							Mission^.JPick			:= WorkArea^[Mission^.PPick].JPick + WorkAreaOffset^[Mission^.PPick].J;
							Mission^.KPick			:= Pallet^[Forming^[WorkAreaState^[Mission^.PPlace].F].Pallet].X; (*+ PickPlaceParameters^.OffsetKPick;*)//Layer^[WorkArea^[Mission^.PPick].Layer].X + PickPlaceParameters^.OffsetKPick;//1150;//Layer^[WorkArea^[cwa].Layer].X + 20; 
							Mission^.KPickTorque	:= KPICKTORQUELAYER;
							Mission^.KPickMode 		:= KSUCTIONMODE;
							Mission^.XPlace			:= WorkArea^[Mission^.PPlace].X + WorkAreaOffset^[Mission^.PPlace].X;
							IF WorkAreaState^[cwa].P = 0 THEN       // se devo depositare la falda sul pallet
								Mission^.YPlace			:= WorkArea^[Mission^.PPlace].Y + WorkAreaOffset^[Mission^.PPlace].Y + (Pallet^[Forming^[WorkAreaState^[Mission^.PPlace].F].Pallet].Y / 2); //!!! Modificato !!!!!//WorkArea^[Mission^.PPlace].Y + (Layer^[Forming^[WorkAreaState^[cwa].F].Layer].Y / 2);
								Mission^.ZPlace			:= WorkArea^[Mission^.PPlace].Z + WorkAreaOffset^[Mission^.PPlace].Z + WorkArea^[Mission^.PPlace].H + Layer^[Forming^[WorkAreaState^[Mission^.PPlace].F].Layer].Z + PickPlaceParameters^.OffsetZPlaceLayer;
							ELSE									// se devo depositare la falda su uno strato di pacchi
								Mission^.YPlace			:= WorkArea^[Mission^.PPlace].Y + WorkAreaOffset^[Mission^.PPlace].Y + (Pallet^[Forming^[WorkAreaState^[Mission^.PPlace].F].Pallet].Y / 2);
								Mission^.ZPlace			:= WorkArea^[Mission^.PPlace].H + Layer^[Forming^[WorkAreaState^[Mission^.PPlace].F].PackXP[WorkAreaState^[Mission^.PPlace].P].Layer].Z + PickPlaceParameters^.OffsetZPlaceLayer;
							END_IF
							Mission^.JPlace			:= WorkArea^[Mission^.PPlace].JPlace + WorkAreaOffset^[Mission^.PPlace].J;
							Mission^.KPlace			:= Mission^.KPick;//WorkArea^[Mission^.PPick].KPick;//Layer^[WorkArea^[cwa].Layer].X + 20;
							Mission^.KPlaceMode 	:= KSUCTIONMODE;
							Mission^.XPlaceApproach	:= Mission^.XPlace;
							Mission^.YPlaceApproach	:= Mission^.YPlace;
							Mission^.ZPlaceApproach	:= Mission^.ZPlace;
							Mission^.JPlaceApproach	:= Mission^.JPlace;
							IF WorkAreaState^[Mission^.PPlace].P = 0 THEN			// se devo depositare la falda sul pallet
								Mission^.XDim			:= Layer^[Forming^[WorkAreaState^[Mission^.PPlace].F].Layer].X;
								Mission^.YDim			:= Layer^[Forming^[WorkAreaState^[Mission^.PPlace].F].Layer].Y;
								Mission^.ZDim			:= Layer^[Forming^[WorkAreaState^[Mission^.PPlace].F].Layer].Z;
							ELSE										// se devo depositare la falda su uno strato di pacchi
								Mission^.XDim			:= Layer^[Forming^[WorkAreaState^[Mission^.PPlace].F].PackXP[WorkAreaState^[Mission^.PPlace].P].Layer].X;
								Mission^.YDim			:= Layer^[Forming^[WorkAreaState^[Mission^.PPlace].F].PackXP[WorkAreaState^[Mission^.PPlace].P].Layer].Y;
								Mission^.ZDim			:= Layer^[Forming^[WorkAreaState^[Mission^.PPlace].F].PackXP[WorkAreaState^[Mission^.PPlace].P].Layer].Z;
							END_IF
							
							WorkAreaManager^.State := WAMANAGER_CICLO_PRELIEVO_FALDA_RUN;
							EXIT;
							
						WAMANAGER_CICLO_PRELIEVO_FALDA_RUN:	
							IF Mission^.State = MISSION_STATE_PRELIEVO_FALDA_RUN THEN
								;
							ELSIF Mission^.State = MISSION_STATE_PRELIEVO_FALDA_END THEN
								WorkAreaManager^.State := WAMANAGER_CICLO_PRELIEVO_FALDA_END;
								EXIT;
							ELSIF Mission^.State = MISSION_STATE_ERROR THEN
								;
							END_IF
	
						WAMANAGER_CICLO_PRELIEVO_FALDA_END:	
							//IF Mission^.TPick = TPICK_LAYER THEN
								IF WorkArea^[Mission^.PPick].Typology = TYPOLOGY_LAYER THEN
									IF WorkArea^[Mission^.PPick].H > WorkArea^[Mission^.PPick].Z + Layer^[WorkArea^[Mission^.PPick].Layer].Z THEN
										WorkArea^[Mission^.PPick].H := ModuleAX_Z^.Ax^.Status.ActPosition; (*- WorkArea^[Mission^.PPick].Z;*)//WorkArea^[Mission^.PPick].H - Layer^[WorkArea^[Mission^.PPick].Layer].Z;
										WorkArea^[Mission^.PPick].DoLearn_Z := 2;
										WorkArea^[Mission^.PPick].Learned_Z := ModuleAX_Z^.Ax^.Status.ActPosition;
									ELSE
										WorkArea^[Mission^.PPick].H := 0;
										WorkArea^[Mission^.PPick].DoLearn_Z := 1;
										WorkArea^[Mission^.PPick].Learned_Z := ALTEZZA_CATASTA_FALDE;
										//WorkAreaState^[Mission^.PPick].State := WORKAREA_STATE_OCCUPIED_ENDED;	
									END_IF
								END_IF
							//END_IF
							WorkAreaManager^.State 	:= WAMANAGER_CICLO_DEPOSITO_FALDA_RUN;
							EXIT;
						
						WAMANAGER_CICLO_DEPOSITO_FALDA_RUN:	
							IF Mission^.State = MISSION_STATE_DEPOSITO_FALDA_RUN THEN
								;
							ELSIF Mission^.State = MISSION_STATE_DEPOSITO_FALDA_END THEN
								RestoreCWA^ := TRUE;
								PreviousPWA^ := pwa;
								WorkAreaManager^.State 	:= WAMANAGER_CICLO_DEPOSITO_FALDA_END;	// setto lo stato del WAMANAGER
								EXIT;
							ELSIF Mission^.State = MISSION_STATE_ERROR THEN
								;
							END_IF
							
						WAMANAGER_CICLO_DEPOSITO_FALDA_END:
							//IF WorkAreaState^[Mission^.PPlace].L = 0 THEN						// se la workarea indica l'assenza della falda
								(* Assegno WorkArea^[cwa].L=1 completamento deposito Falda *)
								WorkAreaState^[Mission^.PPlace].L := 1;							// setto la presenza della falda sulla Piazzola dove depositerò il pallet
								WorkAreaState^[Mission^.PPlace].P := WorkAreaState^[Mission^.PPlace].P + 1; // Aggiorno il numero del pacco successivo che si deve depositare
								(* Aggiorno Altezza Pallet su Layer *)
								IF WorkAreaState^[Mission^.PPlace].P > 0 THEN
									WorkArea^[Mission^.PPlace].H := WorkArea^[cwa].H + Layer^[Forming^[WorkAreaState^[Mission^.PPlace].F].Layer].Z;
								ELSE
									WorkArea^[Mission^.PPlace].HPL := WorkArea^[cwa].HPL + Layer^[Forming^[WorkAreaState^[Mission^.PPlace].F].Layer].Z;
								END_IF
								
								(* Aggiorno il numero del pacco successivo che si deve depositare, se il doposito falda è stato effettuato sopra uno strato di pacchi 
								IF WorkAreaState^[Mission^.PPlace].P > 1 THEN						// doposito falda è stato effettuato sopra uno strato di pacchi
										// Aggiorno il numero del pacco successivo che si deve depositare
								ELSE
									WorkAreaState^[Mission^.PPlace].P := 1;							// Aggiorno il numero del pacco successivo che si deve depositare = pacco n°1
								END_IF*)
								
								(* Controllo Fine Pallettizzazione o Deposito Falda Dopo Strato Layer*)
								(* COME FACCIO A SAPERE SE è L'ULTIMO PACCO ? -> Si controlla la Grip=-1 *)
								(* Per sicurezza le controllo su entrambi le direzioni POSITIVA/NEGATIVA *)
								IF Forming^[WorkAreaState^[Mission^.PPlace].F].PackXP[WorkAreaState^[Mission^.PPlace].P].Grip = -1 OR
									Forming^[WorkAreaState^[Mission^.PPlace].F].PackXN[WorkAreaState^[Mission^.PPlace].P].Grip = -1 THEN
									WorkAreaState^[Mission^.PPlace].State := WORKAREA_STATE_OCCUPIED_WORKED;
								END_IF	
								
								RestoreCWA^ := TRUE;
								PreviousPWA^ := pwa;
								WorkAreaManager^.State 	:= WAMANAGER_NOP;
								EXIT;	
							//ELSE														// non dovrebbe mai accadere
							//	WorkAreaState^[cwa].L := 1;	
							//	WorkAreaState^[cwa].State := WORKAREA_STATE_OCCUPIED_WORKED;
							//	WorkAreaManager^.State 	:= WAMANAGER_NOP;
							//	EXIT;
							//END_IF
							
						(* Creo Missione Pacco *)
						WAMANAGER_CICLO_PACCO_INIT:
							IF cwa = UltimaWAAssegnazionePacco AND cwa<>0 THEN
								(* Reset della memoria utilizzata per forzare il ciclo di riposo in ciclo di prelievo pacco *)
								//ForzaPrelievoPaccoDuranteCicloDiRiposo := FALSE;			
								(* Definisco dse la WORKAREA è negativa o positiva *)
								IF WorkAreaState^[cwa].PN < 0 THEN							// se la Workarea non è stata inizializzata (-1) vado a definire se è a DX o SX del ribaltino
									IF WorkPickPoint^[ppick].Xv < WorkArea^[cwa].X THEN		// Se la quota X è MINORE della quota del ribaltino definisco che la workarea è NEGATIVA 
										WorkAreaState^[cwa].PN := 0;
									ELSE													// Se la quota X è MAGGIORE della quota del ribaltino definisco che la workarea è POSITIVA 
										WorkAreaState^[cwa].PN := 1;
									END_IF
								END_IF
								
								Mission^.PPick := ppick;								   	// Assegno il numero della Punto di prelievo
								Mission^.TPick := TPICK_PACK;							   	// Assegno il tipo di Prelievo
								Mission^.PPlace := cwa;									   	// Assegno il numero della piazzola di deposito
								Mission^.XDim := WorkPickPointState^[Mission^.PPick].XDim; 	// Assegno la dimensione X del pacco presente nel punto di prelievo designato
								Mission^.YDim := WorkPickPointState^[Mission^.PPick].YDim; 	// Assegno la dimensione X del pacco presente nel punto di prelievo designato
								Mission^.ZDim := WorkPickPointState^[Mission^.PPick].ZDim; 	// Assegno la dimensione X del pacco presente nel punto di prelievo designato
								
								(* Definisco il tipo di presa dei pacchi "sinistri" e "destri" *)
								IF WorkAreaState^[cwa].PN = 0 THEN							
									jp := Forming^[WorkAreaState^[cwa].F].PackXP[WorkAreaState^[cwa].P].JP;		// Tipo di presa della pinza
									vo := Forming^[WorkAreaState^[cwa].F].PackXP[WorkAreaState^[cwa].P].Grip;	// Tipo di disposizione del pacco sul ribaltino
								ELSE
									jp := Forming^[WorkAreaState^[cwa].F].PackXN[WorkAreaState^[cwa].P].JP;		// Tipo di presa della pinza
									vo := Forming^[WorkAreaState^[cwa].F].PackXN[WorkAreaState^[cwa].P].Grip;	// Tipo di disposizione del pacco sul ribaltino
								END_IF
								(* Controllo se lo spessore del pacco è minore della lunghezza della pinza *)
								IF Mission^.ZDim < TCPParameter^.Z AND 						// Altezza pacco sul ribaltino < di un parametro
									vo = 1 THEN												// Presa pacco in orrizzontale
									ZOffsetPick 	:= TCPParameter^.Z - Mission^.ZDim;		// Offset da utilizzare successivamente nel calcolo della quota di prelievo
									ZOffsetPlace 	:= TCPParameter^.Z - Mission^.ZDim;		// Offset da utilizzare successivamente nel calcolo della quota di prelievo
								ELSE	
									ZOffsetPick 	:= 0;									// Offset da utilizzare successivamente nel calcolo della quota di prelievo
									ZOffsetPlace 	:= 0;									// Offset da utilizzare successivamente nel calcolo della quota di prelievo
								END_IF
								
								IF vo = 0 THEN 															// Se ho prelievo verticale
									CASE TIPO_RIBALTINO OF
										(* TIPO 1 = RIBALTINO_DOPO_SQUADRO *)
										1: 
											HalfPackDim := Mission^.YDim/2;										// Metà pacco = (dimensione Y)/2
											(* Verticale *)
											IF jp = 1 THEN														// Prelievo lungo X (Longitudinale)
												(* Longitudinale *)
												kpick := Mission^.XDim;										 	// Quota di prelievo Asse K
												torque := Forming^[WorkAreaState^[cwa].F].KLT;					// Valore di coppia Asse K
											ELSE																// Prelievo lungo Y (Trasversale)
												(* Trasversale *)
												kpick := Mission^.ZDim;	//Forming^[WorkAreaState^[cwa].F].PZ;	// Quota di prelievo Asse K
												torque := Forming^[WorkAreaState^[cwa].F].KTT;					// Valore di coppia Asse K
											END_IF
											XPick := WorkPickPoint^[Mission^.PPick].Xv + 		// Quota X Ribaltino
													 WorkPickPointOffset^[Mission^.PPick].Xv;	//Offset Posizione ribaltino in direzione X	
											YPick := WorkPickPoint^[Mission^.PPick].Yv + 		// Quota Y ribaltino
													 WorkPickPointOffset^[Mission^.PPick].Yv + //Offset Posizione ribaltino in direzione Y
													 (Mission^.ZDim / 2);					// (Dimensione pacco Z)/2
											ZPick := WorkPickPoint^[Mission^.PPick].Zv + 	// Quota Z ribaltino
													 WorkPickPointOffset^[Mission^.PPick].Zv + //Offset Posizione ribaltino in direzione Z	
													 Mission^.YDim + 						// Dimensione Y del pacco	
													 Forming^[WorkAreaState^[cwa].F].PIZ + 	// Offset di prelievo dato dalla formatura			
													 WorkPickPointState^[ppick].ZTilter;	// Quota asse ribaltino
											(* In base al tipo di pallettizzatore setto la quota per la presa in modo che i pacchi vengano depositati in modo corretto *)		 		 
											CASE VERSO_PALLETTIZZATORE OF
												PALLETTIZZATORE_DX:
																	JPick := WorkPickPoint^[Mission^.PPick].Jv + 		// Quota rotazione data dalla disposizione del ribaltino
																			 WorkPickPointOffset^[Mission^.PPick].Jv + 	//Offset Posizione ribaltino in direzione Z	
																 			(90 * jp) - 90 +							// Quota rotazione stabilita dal tipo di presa	
																			180;
											
												PALLETTIZZATORE_SX:
																	JPick := WorkPickPoint^[Mission^.PPick].Jv + 	// Quota rotazione data dalla disposizione del ribaltino
																			 WorkPickPointOffset^[Mission^.PPick].Jv + //Offset Posizione ribaltino in direzione Z	
																 			(90 * jp) - 90;								// Quota rotazione stabilita dal tipo di presa								
											END_CASE		 
											(* Differenza tra valori reali e nominali  *)
											DifferenceRealNominalDimensionZ := Mission^.YDim - Forming^[WorkAreaState^[cwa].F].PY;
											(* Valorizzo la variabile che serve per calolare la quota di fuori ingombro verticale della pinza *)
											Dimensione_Z_ElementoInPresaX_Ingombro := Mission^.YDim + Forming^[WorkAreaState^[cwa].F].PIZ;
										(* TIPO 2 = RIBALTINO_DIRETTO *)
										2:
											HalfPackDim := Mission^.ZDim/2;										// Metà pacco = (dimensione Z)/2
											(* Verticale *)
											IF jp = 0 THEN														// Prelievo (Longitudinale)
												(* Longitudinale *)
												kpick := Mission^.ZDim;                                     	// Quota di prelievo Asse K
												torque := Forming^[WorkAreaState^[cwa].F].KLT;					// Valore di coppia Asse K
											ELSE																// Prelievo lungo Y (Trasversale)
												(* Trasversale *)
												kpick := Mission^.YDim;	//Forming^[WorkAreaState^[cwa].F].PZ;	// Quota di prelievo Asse K
												torque := Forming^[WorkAreaState^[cwa].F].KTT;					// Valore di coppia Asse K
											END_IF
											XPick := WorkPickPoint^[Mission^.PPick].Xv + 		// Quota X Ribaltino
													 WorkPickPointOffset^[Mission^.PPick].Xv +	//Offset Posizione ribaltino in direzione X	
													 Mission^.ZDim/2;								// Metà pacco = (dimensione Z) /2
											YPick := WorkPickPoint^[Mission^.PPick].Yv + 		// Quota Y ribaltino
													 WorkPickPointOffset^[Mission^.PPick].Yv;  //Offset Posizione ribaltino in direzione Y
													//(Mission^.ZDim / 2);					// (Dimensione pacco Z)/2
											ZPick := WorkPickPoint^[Mission^.PPick].Zv + 	// Quota Z ribaltino
													 WorkPickPointOffset^[Mission^.PPick].Zv + //Offset Posizione ribaltino in direzione Z	
													 Mission^.XDim + 						// Dimensione Y del pacco	
													 Forming^[WorkAreaState^[cwa].F].PIZ + 	// Offset di prelievo dato dalla formatura			
													 WorkPickPointState^[ppick].ZTilter;	// Quota asse ribaltino
											(* In base al tipo di pallettizzatore setto la quota per la presa in modo che i pacchi vengano depositati in modo corretto *)		 
											CASE VERSO_PALLETTIZZATORE OF
												PALLETTIZZATORE_DX:
																	JPick := WorkPickPoint^[Mission^.PPick].Jv + 	// Quota rotazione data dalla disposizione del ribaltino
																			 WorkPickPointOffset^[Mission^.PPick].Jv + //Offset Posizione ribaltino in direzione Z	
														 					(90 * (1-jp))+								// Quota rotazione stabilita dal tipo di presa	
																			180;										// +180° per fare in modo che il deposito sul pallet sia uguale per le formature con verso del pal DX e SX
												
												PALLETTIZZATORE_SX:	
																	JPick := WorkPickPoint^[Mission^.PPick].Jv + 	// Quota rotazione data dalla disposizione del ribaltino
																			 WorkPickPointOffset^[Mission^.PPick].Jv + //Offset Posizione ribaltino in direzione Z	
														 					(90 * (1-jp));								// Quota rotazione stabilita dal tipo di presa							
											END_CASE
											(* Differenza tra valori reali e nominali  *)
											DifferenceRealNominalDimensionZ := Mission^.XDim - Forming^[WorkAreaState^[cwa].F].PY;
											(* Valorizzo la variabile che serve per calolare la quota di fuori ingombro verticale della pinza *)
											Dimensione_Z_ElementoInPresaX_Ingombro := Mission^.XDim + Forming^[WorkAreaState^[cwa].F].PIZ;
									END_CASE
									
								ELSE																	// Se ho prelievo orrizzontale
									CASE TIPO_RIBALTINO OF
										(* TIPO 1 = RIBALTINO_DOPO_SQUADRO *)
										1:
											HalfPackDim := Mission^.ZDim/2; 									// Metà pacco = (dimensione Z) /2
											(* Orizzontale *)
											IF jp = 1 THEN														// Prelievo TRASVERSALE
												(* Trasversale *)
												kpick := Mission^.XDim; 										 // Quota di prelievo Asse K
												torque := Forming^[WorkAreaState^[cwa].F].KLT;					// Valore di coppia Asse K
											ELSE																// Prelievo lungo Y (Trasversale)
												(* Longitudinale *)							
												kpick := Mission^.YDim; //Forming^[WorkAreaState^[cwa].F].PY;	// Quota di prelievo Asse K
												torque := Forming^[WorkAreaState^[cwa].F].KTT;					// Valore di coppia Asse K
											END_IF
											
											XPick := WorkPickPoint^[Mission^.PPick].Xh +						// Quota X ribaltino
													 WorkPickPointOffset^[Mission^.PPick].Xh; 					// Offset Posizione ribaltino in direzione X	
											YPick := WorkPickPoint^[Mission^.PPick].Yh + 						// Quota Y ribaltino
													 WorkPickPointOffset^[Mission^.PPick].Yh - 					// Offset Posizione ribaltino in direzione Y
													(Mission^.YDim / 2) - 										// (Dimensione pacco Y)/2
													WorkPickPointState^[ppick].ZTilter;							// Quota asse ribaltino
											ZPick := WorkPickPoint^[Mission^.PPick].Zh + 						// Quota Z ribaltino
													 WorkPickPointOffset^[Mission^.PPick].Zh + 					//Offset Posizione ribaltino in direzione Z
													Mission^.ZDim + 											// Dimensione Z pacco
													Forming^[WorkAreaState^[cwa].F].PIZ + 						// Offset di prelievo dato da formatura
													ZOffsetPick;												// Offset calcolato in precedenza
											(* In base al tipo di pallettizzatore setto la quota per la presa in modo che i pacchi vengano depositati in modo corretto *)		
											CASE VERSO_PALLETTIZZATORE OF
												PALLETTIZZATORE_DX:		
																	JPick := WorkPickPoint^[Mission^.PPick].Jh + 						// Quota rotazione data dalla disposizione del ribaltino
																			 WorkPickPointOffset^[Mission^.PPick].Jh + 					//Offset Posizione ribaltino in direzione J
																			(90 * jp)-90+													// Quota rotazione stabilita dal tipo di presa
																			180;										// +180° per fare in modo che il deposito sul pallet sia uguale per le formature con verso del pal DX e SX
												PALLETTIZZATORE_SX:		
																	JPick := WorkPickPoint^[Mission^.PPick].Jh + 						// Quota rotazione data dalla disposizione del ribaltino
																			 WorkPickPointOffset^[Mission^.PPick].Jh + 					//Offset Posizione ribaltino in direzione J
																			(90 * jp)-90;													// Quota rotazione stabilita dal tipo di presa
											END_CASE
											(* Differenza tra valori reali e nominali *)
											DifferenceRealNominalDimensionZ := Mission^.ZDim - Forming^[WorkAreaState^[cwa].F].PZ;		
											(* Valorizzo la variabile che serve per calolare la quota di fuori ingombro verticale della pinza *)
											Dimensione_Z_ElementoInPresaX_Ingombro := Mission^.ZDim + Forming^[WorkAreaState^[cwa].F].PIZ;
										
										(* TIPO 2 = RIBALTINO_DIRETTO *)
										2:
											HalfPackDim := Mission^.YDim/2; 									// Metà pacco = (dimensione Y) /2
											(* Orizzontale *)
											IF jp = 0 THEN														// Prelievo TRASVERSALE
												(* Trasversale *)
												kpick := Mission^.XDim;											// Quota di prelievo Asse K
												torque := Forming^[WorkAreaState^[cwa].F].KLT;					// Valore di coppia Asse K
											ELSE																// Prelievo lungo Y (Trasversale)
												(* Longitudinale *) 							
												kpick := Mission^.YDim; //Forming^[WorkAreaState^[cwa].F].PY;	// Quota di prelievo Asse K
												torque := Forming^[WorkAreaState^[cwa].F].KTT;					// Valore di coppia Asse K
											END_IF
											
											XPick := WorkPickPoint^[Mission^.PPick].Xh +						// Quota X ribaltino
													 WorkPickPointOffset^[Mission^.PPick].Xh - 					// Offset Posizione ribaltino in direzione X	
													 Mission^.XDim/2;												// (Dimensione pacco Y)/2
											YPick := WorkPickPoint^[Mission^.PPick].Yh + 						// Quota Y ribaltino
													 WorkPickPointOffset^[Mission^.PPick].Yh - 					// Offset Posizione ribaltino in direzione Y
													 WorkPickPointState^[ppick].ZTilter;						// Quota asse ribaltino
											ZPick := WorkPickPoint^[Mission^.PPick].Zh + 						// Quota Z ribaltino
													 WorkPickPointOffset^[Mission^.PPick].Zh + 					//Offset Posizione ribaltino in direzione Z
													Mission^.ZDim + 											// Dimensione Z pacco
													Forming^[WorkAreaState^[cwa].F].PIZ + 						// Offset di prelievo dato da formatura
													ZOffsetPick;												// Offset calcolato in precedenza
											(* In base al tipo di pallettizzatore setto la quota per la presa in modo che i pacchi vengano depositati in modo corretto *)		
											CASE VERSO_PALLETTIZZATORE OF
												PALLETTIZZATORE_DX:												
																	JPick := WorkPickPoint^[Mission^.PPick].Jh + 						// Quota rotazione data dalla disposizione del ribaltino
																			 WorkPickPointOffset^[Mission^.PPick].Jh + 					//Offset Posizione ribaltino in direzione J
																			(90 * (1-jp))+												// Quota rotazione stabilita dal tipo di presa
																			180;
												PALLETTIZZATORE_SX:												
																	JPick := WorkPickPoint^[Mission^.PPick].Jh + 						// Quota rotazione data dalla disposizione del ribaltino
																			 WorkPickPointOffset^[Mission^.PPick].Jh + 					//Offset Posizione ribaltino in direzione J
																			(90 * (1-jp));												// Quota rotazione stabilita dal tipo di presa
											END_CASE
																										
											(* Differenza tra valori reali e nominali *)
											DifferenceRealNominalDimensionZ := Mission^.ZDim - Forming^[WorkAreaState^[cwa].F].PZ;		
											(* Valorizzo la variabile che serve per calolare la quota di fuori ingombro verticale della pinza *)
											Dimensione_Z_ElementoInPresaX_Ingombro := Mission^.ZDim + Forming^[WorkAreaState^[cwa].F].PIZ;
									END_CASE
										
								END_IF
								
								Mission^.XPick			:= XPick;
								Mission^.YPick			:= YPick;
								Mission^.ZPick			:= ZPick;
								Mission^.JPick			:= JPick;
								Mission^.JPickLT		:= jp;
								Mission^.JPickVO		:= vo;
								Mission^.KPick			:= kpick;// + OFFSETKPICK;
								Mission^.KPickTorque	:= torque;
								IF NOT SimulazioneSenzaPallet THEN //Se non sono in simulazione utilizzo la presa con coppia
									Mission^.KPickMode 		:= Forming^[WorkAreaState^[cwa].F].KM;		// valorizzazione del tipo di presa in base al tipo scelto nella formatura
								ELSE
									Mission^.KPickMode 		:= KPOSITIONMODE;
									Mission^.KPick			:= kpick + PickPlaceParameters^.OffsetKPickPack;
								END_IF
								(* Set delle variabili per andare al punto di riposo *)
								X_Riposo	:= XPick;
								Y_Riposo	:= YPick;
								J_Riposo	:= JPick;
								K_Riposo	:= kpick;
								Z_Riposo	:= QuotaFuoriIngombro_Z_AVUOTO;
													
								// Tipo di Traiettoria
								// Mission^.Approach		:= Forming^[WorkAreaState^[cwa].F].PackXN[WorkAreaState^[cwa].P].Trajectory;
								(* Valorizzazione nel caso di Piazzole negative*)
								IF WorkAreaState^[cwa].PN = 1 THEN
									Mission^.XPlace			:= 	WorkArea^[Mission^.PPlace].X + 
																WorkAreaOffset^[Mission^.PPlace].X + 
																Forming^[WorkAreaState^[cwa].F].PackXN[WorkAreaState^[cwa].P].X;
									Mission^.YPlace			:=	WorkArea^[Mission^.PPlace].Y + 
																WorkAreaOffset^[Mission^.PPlace].Y + 
																Forming^[WorkAreaState^[cwa].F].PackXN[WorkAreaState^[cwa].P].Y;
									(* Quota di deposito Z con pacco verticale *)	
									CASE TIPO_RIBALTINO OF

										RIBALTINO_DOPO_SQUADRO:
											IF vo = 0 THEN 							
												Mission^.ZPlace			:= 	//WorkArea^[Mission^.PPlace].Z + 
																			Forming^[WorkAreaState^[cwa].F].PackXN[WorkAreaState^[cwa].P].Z + 
																			Forming^[WorkAreaState^[cwa].F].PLZ + 
																			Forming^[WorkAreaState^[cwa].F].PIZ +
																			WorkArea^[Mission^.PPlace].HPL + 
																			HalfPackDim + 
																			ZOffsetPlace + 
																			PickPlaceParameters^.OffsetZPlacePaccoVerticale +
																			DifferenceRealNominalDimensionZ/2;
											(* Quota di deposito Z con pacco orrizontale *)	
											ELSE
												Mission^.ZPlace			:= 	//WorkArea^[Mission^.PPlace].Z + 
																			Forming^[WorkAreaState^[cwa].F].PackXN[WorkAreaState^[cwa].P].Z + 
																			Forming^[WorkAreaState^[cwa].F].PLZ + 
																			WorkArea^[Mission^.PPlace].HPL + 
																			HalfPackDim + 
																			ZOffsetPlace + 
																			PickPlaceParameters^.OffsetZPlacePaccoOrrizzontale;
																			//DifferenceRealNominalDimensionZ/2;
											END_IF
									
										RIBALTINO_DIRETTO:
											IF vo = 0 THEN 							
												Mission^.ZPlace			:= 	//WorkArea^[Mission^.PPlace].Z + 
																			Forming^[WorkAreaState^[cwa].F].PackXN[WorkAreaState^[cwa].P].Z + 
																			Forming^[WorkAreaState^[cwa].F].PLZ + 
																			Forming^[WorkAreaState^[cwa].F].PIZ +
																			WorkArea^[Mission^.PPlace].HPL + 
																			Mission^.XDiM/2 + 
																			ZOffsetPlace + 
																			PickPlaceParameters^.OffsetZPlacePaccoVerticale +
																			DifferenceRealNominalDimensionZ/2;
											(* Quota di deposito Z con pacco orrizontale *)	
											ELSE
												Mission^.ZPlace			:= 	//WorkArea^[Mission^.PPlace].Z + 
																			Forming^[WorkAreaState^[cwa].F].PackXN[WorkAreaState^[cwa].P].Z + 
																			Forming^[WorkAreaState^[cwa].F].PLZ + 
																			WorkArea^[Mission^.PPlace].HPL + 
																			Mission^.ZDim/2 + 
																			ZOffsetPlace + 
																			PickPlaceParameters^.OffsetZPlacePaccoOrrizzontale +
																			DifferenceRealNominalDimensionZ/2;
											END_IF
									END_CASE
									
									//Mission^.ZPlace			:= WorkArea^[Mission^.PPlace].Z + Forming^[WorkAreaState^[cwa].F].PackXP[WorkAreaState^[cwa].P].Z*2 + WorkArea^[Mission^.PPlace].H;
									CASE Jp OF
										-1:;
										//Presa trasversale	
										0: 
											IF Forming^[WorkAreaState^[cwa].F].PackXN[WorkAreaState^[cwa].P].J = 0 AND TIPO_RIBALTINO = RIBALTINO_DIRETTO THEN
												Mission^.JPlace	:= 	WorkArea^[Mission^.PPlace].J + 
																	WorkAreaOffset^[Mission^.PPlace].J + 
																	Forming^[WorkAreaState^[cwa].F].PackXN[WorkAreaState^[cwa].P].J;																		
											ELSIF Forming^[WorkAreaState^[cwa].F].PackXN[WorkAreaState^[cwa].P].J = 90 AND TIPO_RIBALTINO = RIBALTINO_DIRETTO THEN
												Mission^.JPlace	:= 	WorkArea^[Mission^.PPlace].J + 
																	WorkAreaOffset^[Mission^.PPlace].J + 
																	Forming^[WorkAreaState^[cwa].F].PackXN[WorkAreaState^[cwa].P].J + 90;	
											ELSIF Forming^[WorkAreaState^[cwa].F].PackXN[WorkAreaState^[cwa].P].J = 180 AND TIPO_RIBALTINO = RIBALTINO_DIRETTO THEN
												Mission^.JPlace	:= 	WorkArea^[Mission^.PPlace].J + 
																	WorkAreaOffset^[Mission^.PPlace].J + 
																	Forming^[WorkAreaState^[cwa].F].PackXN[WorkAreaState^[cwa].P].J + 90;
											ELSIF Forming^[WorkAreaState^[cwa].F].PackXN[WorkAreaState^[cwa].P].J = 270 AND TIPO_RIBALTINO = RIBALTINO_DIRETTO THEN
												Mission^.JPlace	:= 	WorkArea^[Mission^.PPlace].J + 
																	WorkAreaOffset^[Mission^.PPlace].J;
											ELSE
												Mission^.JPlace	:= 	WorkArea^[Mission^.PPlace].J + 
																	WorkAreaOffset^[Mission^.PPlace].J + 
																	Forming^[WorkAreaState^[cwa].F].PackXN[WorkAreaState^[cwa].P].J;											
											END_IF
											
											
										//Presa longitudinale
										1:
											CASE VERSO_PALLETTIZZATORE OF 
												
												PALLETTIZZATORE_DX:
													Mission^.JPlace			:= 	WorkArea^[Mission^.PPlace].J + 
																WorkAreaOffset^[Mission^.PPlace].J + 
																Forming^[WorkAreaState^[cwa].F].PackXN[WorkAreaState^[cwa].P].J;
																
												PALLETTIZZATORE_SX:
													Mission^.JPlace			:= 	WorkArea^[Mission^.PPlace].J + 
																WorkAreaOffset^[Mission^.PPlace].J + 
																Forming^[WorkAreaState^[cwa].F].PackXN[WorkAreaState^[cwa].P].J;

											END_CASE
												(*Mission^.JPlace			:= 	WorkArea^[Mission^.PPlace].J + 
																	WorkAreaOffset^[Mission^.PPlace].J + 
																	Forming^[WorkAreaState^[cwa].F].PackXN[WorkAreaState^[cwa].P].J;*)	
																
																				
									END_CASE
									
									IF NOT SimulazioneSenzaPallet THEN //Se non sono in simulazione utilizzo la presa con coppia							
										Mission^.KPlace			:= 	kpick; (*+ 
																PickPlaceParameters^.OffsetKPlacePack;*) // Aggiungere Eventuale Offset x Apertura e Rilascio
									ELSE
										Mission^.KPlace			:= 	kpick + PickPlaceParameters^.OffsetKPickPack;
									END_IF
									Mission^.KPlaceMode 	:= 	Forming^[WorkAreaState^[cwa].F].KM;// KTORQUEMODE;
									(* Quota di Approccio con pacco verticale *)							
									IF (vo = 0 AND DisabilitaApproccioPacciOrrizzontali) OR NOT DisabilitaApproccioPacciOrrizzontali THEN 
										IF  Forming^[WorkAreaState^[cwa].F].PackXN[WorkAreaState^[cwa].P].Trajectory = 0 THEN //NO APPROCCIO
											Mission^.XPlaceApproach	:= Mission^.XPlace;
											Mission^.YPlaceApproach	:= Mission^.YPlace;
											Mission^.ZPlaceApproach	:= Mission^.ZPlace;
											Mission^.JPlaceApproach	:= Mission^.JPlace;
										ELSIF Forming^[WorkAreaState^[cwa].F].PackXN[WorkAreaState^[cwa].P].Trajectory = 1 THEN // APPROCCIO STANDARD
											Mission^.XPlaceApproach	:= 	Mission^.XPlace + 
																		Forming^[WorkAreaState^[cwa].F].AX;
											Mission^.YPlaceApproach	:= 	Mission^.YPlace - 
																		Forming^[WorkAreaState^[cwa].F].AY;
											Mission^.ZPlaceApproach	:= 	Mission^.ZPlace + 
																		Forming^[WorkAreaState^[cwa].F].AZ;
											Mission^.JPlaceApproach	:= 	Mission^.JPlace;
										ELSIF Forming^[WorkAreaState^[cwa].F].PackXN[WorkAreaState^[cwa].P].Trajectory = 111 THEN // APPROCCIO STANDARD
											Mission^.XPlaceApproach	:= 	Mission^.XPlace + 
																		Forming^[WorkAreaState^[cwa].F].AX;
											Mission^.YPlaceApproach	:= 	Mission^.YPlace - 
																		Forming^[WorkAreaState^[cwa].F].AY;
											Mission^.ZPlaceApproach	:= 	Mission^.ZPlace + 
																		Forming^[WorkAreaState^[cwa].F].AZ;
											Mission^.JPlaceApproach	:= 	Mission^.JPlace;
										ELSIF Forming^[WorkAreaState^[cwa].F].PackXN[WorkAreaState^[cwa].P].Trajectory = 2	THEN // ESTERNO-INTERNO X
											Mission^.XPlaceApproach	:= 	Mission^.XPlace - 
																		Forming^[WorkAreaState^[cwa].F].AX;
											Mission^.YPlaceApproach	:= 	Mission^.YPlace - 	
																		Forming^[WorkAreaState^[cwa].F].AY;
											Mission^.ZPlaceApproach	:= 	Mission^.ZPlace + 
																		Forming^[WorkAreaState^[cwa].F].AZ;
											Mission^.JPlaceApproach	:= 	Mission^.JPlace;
										ELSIF Forming^[WorkAreaState^[cwa].F].PackXN[WorkAreaState^[cwa].P].Trajectory = 101	THEN // ESTERNO-INTERNO X
											Mission^.XPlaceApproach	:= 	Mission^.XPlace - 
																		Forming^[WorkAreaState^[cwa].F].AX;
											Mission^.YPlaceApproach	:= 	Mission^.YPlace - 	
																		Forming^[WorkAreaState^[cwa].F].AY;
											Mission^.ZPlaceApproach	:= 	Mission^.ZPlace + 
																		Forming^[WorkAreaState^[cwa].F].AZ;
											Mission^.JPlaceApproach	:= 	Mission^.JPlace;
										ELSIF Forming^[WorkAreaState^[cwa].F].PackXN[WorkAreaState^[cwa].P].Trajectory = 201	THEN // ESTERNO-INTERNO X
											Mission^.XPlaceApproach	:= 	Mission^.XPlace + 
																		Forming^[WorkAreaState^[cwa].F].AX;
											Mission^.YPlaceApproach	:= 	Mission^.YPlace - 	
																		Forming^[WorkAreaState^[cwa].F].AY;
											Mission^.ZPlaceApproach	:= 	Mission^.ZPlace + 
																		Forming^[WorkAreaState^[cwa].F].AZ;
											Mission^.JPlaceApproach	:= 	Mission^.JPlace;
										ELSIF Forming^[WorkAreaState^[cwa].F].PackXN[WorkAreaState^[cwa].P].Trajectory = 3	THEN //
											Mission^.XPlaceApproach	:= 	Mission^.XPlace + 
																		Forming^[WorkAreaState^[cwa].F].AX;
											Mission^.YPlaceApproach	:= 	Mission^.YPlace + 
																		Forming^[WorkAreaState^[cwa].F].AY;
											Mission^.ZPlaceApproach	:= 	Mission^.ZPlace + 
																		Forming^[WorkAreaState^[cwa].F].AZ;
											Mission^.JPlaceApproach	:= 	Mission^.JPlace;	
										ELSIF Forming^[WorkAreaState^[cwa].F].PackXN[WorkAreaState^[cwa].P].Trajectory = 4	THEN // NON USATO
											Mission^.XPlaceApproach	:= 	Mission^.XPlace - 
																		Forming^[WorkAreaState^[cwa].F].AX;
											Mission^.YPlaceApproach	:= 	Mission^.YPlace + 
																		Forming^[WorkAreaState^[cwa].F].AY;
											Mission^.ZPlaceApproach	:= 	Mission^.ZPlace + 
																		Forming^[WorkAreaState^[cwa].F].AZ;
											Mission^.JPlaceApproach	:= 	Mission^.JPlace;
										ELSIF Forming^[WorkAreaState^[cwa].F].PackXN[WorkAreaState^[cwa].P].Trajectory = 5 THEN	//Esterno-Interno Direzione Y !!!!!!!!! modificare con 11 e 21
											Mission^.XPlaceApproach	:= 	Mission^.XPlace;
											IF (Mission^.JPlace = 90 OR Mission^.JPlace = 270) AND Mission^.YPlace >= (WorkArea^[Mission^.PPlace].Y + Pallet^[Workarea^[Mission^.PPlace].Pallet].Y/2) THEN
												Mission^.YPlaceApproach	:= 	Mission^.YPlace + 
																		Forming^[WorkAreaState^[cwa].F].AY;
											ELSE //NORD
												Mission^.YPlaceApproach	:= 	Mission^.YPlace - 
																		Forming^[WorkAreaState^[cwa].F].AY;
											END_IF
											
											Mission^.ZPlaceApproach	:= 	Mission^.ZPlace +
																		Forming^[WorkAreaState^[cwa].F].AZ;
											Mission^.JPlaceApproach	:= 	Mission^.JPlace; 
										ELSIF Forming^[WorkAreaState^[cwa].F].PackXN[WorkAreaState^[cwa].P].Trajectory = 11 THEN	//Esterno-Interno Direzione Y !!!!!!!!! modificare con 11 e 21
											Mission^.XPlaceApproach	:= 	Mission^.XPlace;
											IF (Mission^.JPlace = 90 OR Mission^.JPlace = 270) AND Mission^.YPlace >= (WorkArea^[Mission^.PPlace].Y + Pallet^[Workarea^[Mission^.PPlace].Pallet].Y/2) THEN
												Mission^.YPlaceApproach	:= 	Mission^.YPlace + 
																		Forming^[WorkAreaState^[cwa].F].AY;
											ELSE
												Mission^.YPlaceApproach	:= 	Mission^.YPlace - 
																		Forming^[WorkAreaState^[cwa].F].AY;
											END_IF
											
											Mission^.ZPlaceApproach	:= 	Mission^.ZPlace +
																		Forming^[WorkAreaState^[cwa].F].AZ;
											Mission^.JPlaceApproach	:= 	Mission^.JPlace; 	
										ELSIF Forming^[WorkAreaState^[cwa].F].PackXN[WorkAreaState^[cwa].P].Trajectory = 21 THEN	//Esterno-Interno Direzione Y e BASTA!!!!!!!!! modificare con 11 e 21
											Mission^.XPlaceApproach	:= 	Mission^.XPlace;
											IF (Mission^.JPlace = 90 OR Mission^.JPlace = 270) AND Mission^.YPlace >= (WorkArea^[Mission^.PPlace].Y + Pallet^[Workarea^[Mission^.PPlace].Pallet].Y/2) THEN
												Mission^.YPlaceApproach	:= 	Mission^.YPlace + 
																		Forming^[WorkAreaState^[cwa].F].AY;
											ELSE
												Mission^.YPlaceApproach	:= 	Mission^.YPlace - 
																		Forming^[WorkAreaState^[cwa].F].AY;
											END_IF
											
											Mission^.ZPlaceApproach	:= 	Mission^.ZPlace +
																		Forming^[WorkAreaState^[cwa].F].AZ;
											Mission^.JPlaceApproach	:= 	Mission^.JPlace; 	
										END_IF
									ELSIF DisabilitaApproccioPacciOrrizzontali AND vo = 1 THEN
										Mission^.XPlaceApproach	:= Mission^.XPlace;
										Mission^.YPlaceApproach	:= Mission^.YPlace;
										Mission^.ZPlaceApproach	:= Mission^.ZPlace;
										Mission^.JPlaceApproach	:= Mission^.JPlace;	
									END_IF
								
								ELSE (* Valorizzazione nel caso di Piazzole positive *)
									Mission^.XPlace			:= 	WorkArea^[Mission^.PPlace].X + 
																WorkAreaOffset^[Mission^.PPlace].X + 
																Forming^[WorkAreaState^[cwa].F].PackXP[WorkAreaState^[cwa].P].X;
									Mission^.YPlace			:= 	WorkArea^[Mission^.PPlace].Y + 
																WorkAreaOffset^[Mission^.PPlace].Y + 
																Forming^[WorkAreaState^[cwa].F].PackXP[WorkAreaState^[cwa].P].Y;
									
									(* Quota di deposito Z con pacco verticale *)	
									CASE TIPO_RIBALTINO OF

										RIBALTINO_DOPO_SQUADRO:
											IF vo = 0 THEN 							
												Mission^.ZPlace			:= 	//WorkArea^[Mission^.PPlace].Z + 
																			Forming^[WorkAreaState^[cwa].F].PackXP[WorkAreaState^[cwa].P].Z + 
																			Forming^[WorkAreaState^[cwa].F].PLZ + 
																			Forming^[WorkAreaState^[cwa].F].PIZ +
																			WorkArea^[Mission^.PPlace].HPL + 
																			HalfPackDim + 
																			ZOffsetPlace + 
																			PickPlaceParameters^.OffsetZPlacePaccoVerticale +
																			DifferenceRealNominalDimensionZ/2;
											(* Quota di deposito Z con pacco orrizontale *)	
											ELSE
												Mission^.ZPlace			:= 	//WorkArea^[Mission^.PPlace].Z + 
																			Forming^[WorkAreaState^[cwa].F].PackXP[WorkAreaState^[cwa].P].Z + 
																			Forming^[WorkAreaState^[cwa].F].PLZ + 
																			WorkArea^[Mission^.PPlace].HPL + 
																			HalfPackDim + 
																			ZOffsetPlace + 
																			PickPlaceParameters^.OffsetZPlacePaccoOrrizzontale;
																			//DifferenceRealNominalDimensionZ/2;
											END_IF
									
										RIBALTINO_DIRETTO:
											IF vo = 0 THEN 							
												Mission^.ZPlace			:= 	//WorkArea^[Mission^.PPlace].Z + 
																			Forming^[WorkAreaState^[cwa].F].PackXP[WorkAreaState^[cwa].P].Z + 
																			Forming^[WorkAreaState^[cwa].F].PLZ + 
																			Forming^[WorkAreaState^[cwa].F].PIZ +
																			WorkArea^[Mission^.PPlace].HPL + 
																			Mission^.XDiM/2 + 
																			ZOffsetPlace + 
																			PickPlaceParameters^.OffsetZPlacePaccoVerticale +
																			DifferenceRealNominalDimensionZ/2;
											(* Quota di deposito Z con pacco orrizontale *)	
											ELSE
												Mission^.ZPlace			:= 	//WorkArea^[Mission^.PPlace].Z + 
																			Forming^[WorkAreaState^[cwa].F].PackXP[WorkAreaState^[cwa].P].Z + 
																			Forming^[WorkAreaState^[cwa].F].PLZ + 
																			WorkArea^[Mission^.PPlace].HPL + 
																			Mission^.ZDim/2 + 
																			ZOffsetPlace + 
																			PickPlaceParameters^.OffsetZPlacePaccoOrrizzontale +
																			DifferenceRealNominalDimensionZ/2;
											END_IF
									END_CASE
									//Mission^.ZPlace			:= WorkArea^[Mission^.PPlace].Z + Forming^[WorkAreaState^[cwa].F].PackXN[WorkAreaState^[cwa].P].Z*2 + WorkArea^[Mission^.PPlace].H;
									Mission^.JPlace			:= 	WorkArea^[Mission^.PPlace].J + 
																WorkAreaOffset^[Mission^.PPlace].J + 
																Forming^[WorkAreaState^[cwa].F].PackXP[WorkAreaState^[cwa].P].J-
																(90*(1-JP)); //x deposito con prelievo TRASVERSALE
									CASE VERSO_PALLETTIZZATORE OF 
										
										PALLETTIZZATORE_DX:
											Mission^.JPlace	:= 	WorkArea^[Mission^.PPlace].J + 
																WorkAreaOffset^[Mission^.PPlace].J + 
																Forming^[WorkAreaState^[cwa].F].PackXP[WorkAreaState^[cwa].P].J-
																(90*(1-JP));
														
										PALLETTIZZATORE_SX:
											Mission^.JPlace	:= 	WorkArea^[Mission^.PPlace].J + 
																WorkAreaOffset^[Mission^.PPlace].J + 
																Forming^[WorkAreaState^[cwa].F].PackXP[WorkAreaState^[cwa].P].J-
																(90*(1-JP));

									END_CASE							
																
																
									IF NOT SimulazioneSenzaPallet THEN //Se non sono in simulazione utilizzo la presa con coppia							
										Mission^.KPlace			:= 	kpick; (*+ 
																PickPlaceParameters^.OffsetKPlacePack;*) // Aggiungere Eventuale Offset x Apertura e Rilascio
									ELSE
										Mission^.KPlace			:= 	kpick + PickPlaceParameters^.OffsetKPickPack;
									END_IF
									Mission^.KPlaceMode 	:= 	KTORQUEMODE;
									(* Quota di Approccio con pacco verticale *)							
									IF (vo = 0 AND DisabilitaApproccioPacciOrrizzontali) OR NOT DisabilitaApproccioPacciOrrizzontali THEN 
										IF  Forming^[WorkAreaState^[cwa].F].PackXP[WorkAreaState^[cwa].P].Trajectory = 0 THEN
											Mission^.XPlaceApproach	:= Mission^.XPlace;
											Mission^.YPlaceApproach	:= Mission^.YPlace;
											Mission^.ZPlaceApproach	:= Mission^.ZPlace;
											Mission^.JPlaceApproach	:= Mission^.JPlace;
										ELSIF  Forming^[WorkAreaState^[cwa].F].PackXP[WorkAreaState^[cwa].P].Trajectory = 1 THEN	
											Mission^.XPlaceApproach	:= 	Mission^.XPlace - 
																		Forming^[WorkAreaState^[cwa].F].AX;
											Mission^.YPlaceApproach	:= 	Mission^.YPlace - 
																		Forming^[WorkAreaState^[cwa].F].AY;
											Mission^.ZPlaceApproach	:= 	Mission^.ZPlace + 
																		Forming^[WorkAreaState^[cwa].F].AZ;
											Mission^.JPlaceApproach	:= 	Mission^.JPlace;
										ELSIF  Forming^[WorkAreaState^[cwa].F].PackXP[WorkAreaState^[cwa].P].Trajectory = 111 THEN	
											Mission^.XPlaceApproach	:= 	Mission^.XPlace - 
																		Forming^[WorkAreaState^[cwa].F].AX;
											Mission^.YPlaceApproach	:= 	Mission^.YPlace - 
																		Forming^[WorkAreaState^[cwa].F].AY;
											Mission^.ZPlaceApproach	:= 	Mission^.ZPlace + 
																		Forming^[WorkAreaState^[cwa].F].AZ;
											Mission^.JPlaceApproach	:= 	Mission^.JPlace;
										ELSIF  Forming^[WorkAreaState^[cwa].F].PackXP[WorkAreaState^[cwa].P].Trajectory = 2 THEN	
											Mission^.XPlaceApproach	:= 	Mission^.XPlace + 
																		Forming^[WorkAreaState^[cwa].F].AX;
											Mission^.YPlaceApproach	:= 	Mission^.YPlace - 
																		Forming^[WorkAreaState^[cwa].F].AY;
											Mission^.ZPlaceApproach	:= 	Mission^.ZPlace + 
																		Forming^[WorkAreaState^[cwa].F].AZ;
											Mission^.JPlaceApproach	:= 	Mission^.JPlace;
										ELSIF  Forming^[WorkAreaState^[cwa].F].PackXP[WorkAreaState^[cwa].P].Trajectory = 101 THEN	
											Mission^.XPlaceApproach	:= 	Mission^.XPlace + 
																		Forming^[WorkAreaState^[cwa].F].AX;
											Mission^.YPlaceApproach	:= 	Mission^.YPlace - 
																		Forming^[WorkAreaState^[cwa].F].AY;
											Mission^.ZPlaceApproach	:= 	Mission^.ZPlace + 
																		Forming^[WorkAreaState^[cwa].F].AZ;
											Mission^.JPlaceApproach	:= 	Mission^.JPlace;
										ELSIF  Forming^[WorkAreaState^[cwa].F].PackXP[WorkAreaState^[cwa].P].Trajectory = 101 THEN	
											Mission^.XPlaceApproach	:= 	Mission^.XPlace + 
																		Forming^[WorkAreaState^[cwa].F].AX;
											Mission^.YPlaceApproach	:= 	Mission^.YPlace - 
																		Forming^[WorkAreaState^[cwa].F].AY;
											Mission^.ZPlaceApproach	:= 	Mission^.ZPlace + 
																		Forming^[WorkAreaState^[cwa].F].AZ;
											Mission^.JPlaceApproach	:= 	Mission^.JPlace;
										ELSIF  Forming^[WorkAreaState^[cwa].F].PackXP[WorkAreaState^[cwa].P].Trajectory = 201 THEN	
											Mission^.XPlaceApproach	:= 	Mission^.XPlace - 
																		Forming^[WorkAreaState^[cwa].F].AX;
											Mission^.YPlaceApproach	:= 	Mission^.YPlace + 
																		Forming^[WorkAreaState^[cwa].F].AY;
											Mission^.ZPlaceApproach	:= 	Mission^.ZPlace + 
																		Forming^[WorkAreaState^[cwa].F].AZ;
											Mission^.JPlaceApproach	:= 	Mission^.JPlace;	
										ELSIF  Forming^[WorkAreaState^[cwa].F].PackXP[WorkAreaState^[cwa].P].Trajectory = 4 THEN	
											Mission^.XPlaceApproach	:= 	Mission^.XPlace + 
																		Forming^[WorkAreaState^[cwa].F].AX;
											Mission^.YPlaceApproach	:= 	Mission^.YPlace + 
																		Forming^[WorkAreaState^[cwa].F].AY;
											Mission^.ZPlaceApproach	:= 	Mission^.ZPlace + 
																		Forming^[WorkAreaState^[cwa].F].AZ;
											Mission^.JPlaceApproach	:= 	Mission^.JPlace;
										ELSIF Forming^[WorkAreaState^[cwa].F].PackXP[WorkAreaState^[cwa].P].Trajectory = 5 THEN	//Esterno-Interno Direzione Y !!!!!!!!!
											Mission^.XPlaceApproach	:= 	Mission^.XPlace;
											IF (Mission^.JPlace = 90 OR Mission^.JPlace = 270) AND Mission^.YPlace >= (WorkArea^[Mission^.PPlace].Y + Pallet^[Workarea^[Mission^.PPlace].Pallet].Y/2) THEN
												Mission^.YPlaceApproach	:= 	Mission^.YPlace + 
																		Forming^[WorkAreaState^[cwa].F].AY;
											ELSE
												Mission^.YPlaceApproach	:= 	Mission^.YPlace - 
																		Forming^[WorkAreaState^[cwa].F].AY;
											END_IF
											Mission^.ZPlaceApproach	:= 	Mission^.ZPlace;
											Mission^.JPlaceApproach	:= 	Mission^.JPlace; 
										ELSIF Forming^[WorkAreaState^[cwa].F].PackXP[WorkAreaState^[cwa].P].Trajectory = 11 THEN	//Esterno-Interno Direzione Y !!!!!!!!!
											Mission^.XPlaceApproach	:= 	Mission^.XPlace;
											IF (Mission^.JPlace = 90 OR Mission^.JPlace = 270) AND Mission^.YPlace >= (WorkArea^[Mission^.PPlace].Y + Pallet^[Workarea^[Mission^.PPlace].Pallet].Y/2) THEN
												Mission^.YPlaceApproach	:= 	Mission^.YPlace + 
																		Forming^[WorkAreaState^[cwa].F].AY;
											ELSE
												Mission^.YPlaceApproach	:= 	Mission^.YPlace - 
																		Forming^[WorkAreaState^[cwa].F].AY;
											END_IF
											Mission^.ZPlaceApproach	:= 	Mission^.ZPlace;
											Mission^.JPlaceApproach	:= 	Mission^.JPlace;
										ELSIF Forming^[WorkAreaState^[cwa].F].PackXP[WorkAreaState^[cwa].P].Trajectory = 21 THEN	//Esterno-Interno Direzione Y !!!!!!!!!
											Mission^.XPlaceApproach	:= 	Mission^.XPlace;
											IF (Mission^.JPlace = 90 OR Mission^.JPlace = 270) AND Mission^.YPlace >= (WorkArea^[Mission^.PPlace].Y + Pallet^[Workarea^[Mission^.PPlace].Pallet].Y/2) THEN
												Mission^.YPlaceApproach	:= 	Mission^.YPlace + 
																		Forming^[WorkAreaState^[cwa].F].AY;
											ELSE
												Mission^.YPlaceApproach	:= 	Mission^.YPlace - 
																		Forming^[WorkAreaState^[cwa].F].AY;
											END_IF
											Mission^.ZPlaceApproach	:= 	Mission^.ZPlace;
											Mission^.JPlaceApproach	:= 	Mission^.JPlace;
										END_IF	
									ELSIF DisabilitaApproccioPacciOrrizzontali and vo = 1 THEN
										Mission^.XPlaceApproach	:= Mission^.XPlace;
										Mission^.YPlaceApproach	:= Mission^.YPlace;
										IF NOT AbilitaDepositoPaccoOrrizzonataleConTasteggio^ THEN
											Mission^.ZPlaceApproach	:= Mission^.ZPlace;
										ELSE
											Mission^.ZPlaceApproach	:= Mission^.ZPlace + QuotaFittizziaPerTasteggioDepPacchi;
										END_IF
										
										Mission^.JPlaceApproach	:= Mission^.JPlace;	
									END_IF
								END_IF
								(* Setto l'uscita che mi determina il deposito del primo pacco in lenta *)
								IF WorkArea^[Mission^.PPlace].Slow = 1 THEN
									DepositoPaccoInLenta := TRUE;
								END_IF
								
								
								WorkAreaManager^.State 	:= WAMANAGER_CICLO_PRELIEVO_PACCO_RUN;
								WAAssegnazionePaccoNONok := FALSE;
							ELSE
								WAAssegnazionePaccoNONok := TRUE;
							END_IF
							
						WAMANAGER_CICLO_PRELIEVO_PACCO_RUN:
							IF Mission^.State = MISSION_STATE_PRELIEVO_PACCO_RUN THEN
								;
							ELSIF Mission^.State = MISSION_STATE_PRELIEVO_PACCO_END THEN
								WorkAreaManager^.State 	:= WAMANAGER_CICLO_PRELIEVO_PACCO_END;
							ELSIF Mission^.State = MISSION_STATE_ERROR THEN
								;
							ELSIF Mission^.State = MISSION_STATE_NOP AND (NOT HandlingRun OR WorkPickPointState^[Mission^.PPick].TS <> WorkPickPointState^[Mission^.PPick].TC) THEN
								WorkAreaManager^.State 	:= WAMANAGER_NOP;
							END_IF	
						
						WAMANAGER_CICLO_PRELIEVO_PACCO_END:	
							(* Copio Info Pacco da Ribaltino a Pinza *)
							Mission^.Pack := TilterPack^;
							RestoreCWA^ := TRUE;
							PreviousPWA^ := pwa;
							//TFPalletizerSetWPPState(WorkPickPointState,Mission^.PPick,WORKPICKPOINT_PRODOTTO_ASSENTE);
							WorkAreaManager^.State 	:= WAMANAGER_CICLO_DEPOSITO_PACCO_RUN;
							ForzaPrelievoPaccoDuranteCicloDiRiposo := FALSE;	
							
						WAMANAGER_CICLO_DEPOSITO_PACCO_RUN:	
							IF Mission^.State = MISSION_STATE_DEPOSITO_PACCO_RUN THEN
								;
							ELSIF Mission^.State = MISSION_STATE_DEPOSITO_PACCO_END THEN
								RestoreCWA^ := TRUE;
								PreviousPWA^ := pwa;
								WorkAreaManager^.State 	:= WAMANAGER_CICLO_DEPOSITO_PACCO_END;	// setto lo stato del WAMANAGER
							END_IF
						
						WAMANAGER_CICLO_DEPOSITO_PACCO_END:
						
							(* Se era settata la velocità lenta di deposito pacco, questa viene resettata *)
							IF WorkArea^[Mission^.PPlace].Slow = 1 THEN
								WorkArea^[Mission^.PPlace].Slow := 0;
								DepositoPaccoInLenta := FALSE;
							END_IF
						
							IF Mission^.TPick = TPICK_PACK THEN
								FOR i:=1 TO MAXHANDLINGSTACK DO
									WorkAreaState^[Mission^.PPlace].Pack[WorkAreaState^[Mission^.PPlace].P,i] := Mission^.Pack[i];
								END_FOR	
							END_IF
						
							(* Punto alla tabella Formatura per verificare se dopo questo pacco devo gestire una Falda *)
							(* La fine formatura la verifico con i dati -1 *)
							IF Forming^[WorkAreaState^[Mission^.PPlace].F].PackXP[WorkAreaState^[Mission^.PPlace].P].Layer > 0 THEN			// se dopo aver depositato un pacco, questo richiede il deposito di una falda (.Layer > 0)
								WorkAreaState^[Mission^.PPlace].L := 0;															// metto a 0 lo stato del layer della piazzola in modo che il manager al ciclo successivo si acorg che bisogna compiere un ciclo falda
								(* Aggiorno Altezza Pallet su Ultimo Pacco *)
								IF Mission^.TPick = TPICK_PACK THEN													// Controllo che la missione  appena eseguita era un prelievo pacco ( dovrebbe sempre essere così!! mantenuto da vecchia gestione..)
									CASE TIPO_RIBALTINO OF
										RIBALTINO_DOPO_SQUADRO:
											IF Forming^[WorkAreaState^[Mission^.PPlace].F].PackXP[WorkAreaState^[Mission^.PPlace].P].Grip = 0 THEN	// Aggiornamento altezza pallet con pacco in verticale (si considera la dimensione Y del pacco) 
												WorkArea^[Mission^.PPlace].H := WorkArea^[Mission^.PPlace].HPL +												// Altezza pallet + layers utilizzati
																	Forming^[WorkAreaState^[Mission^.PPlace].F].PackXP[WorkAreaState^[Mission^.PPlace].P].Z + 	// Quota "Z" del centro del pacco sulla piazzola, cioè altezza assoluta del baricentro
																	Mission^.YDim/2;													//Dimensione Y /2, indica la distanza dal baricentro al bordo superiore del pacco
											ELSIF Forming^[WorkAreaState^[cwa].F].PackXP[WorkAreaState^[cwa].P].Grip = 1 THEN
												WorkArea^[Mission^.PPlace].H := WorkArea^[Mission^.PPlace].HPL + 												// Altezza pallet + layers utilizzati
																	Forming^[WorkAreaState^[Mission^.PPlace].F].PackXP[WorkAreaState^[Mission^.PPlace].P].Z + 	// Quota "Z" del centro del pacco sulla piazzola, cioè altezza assoluta del baricentro
																	Mission^.ZDim/2;													//Dimensione Z /2, indica la distanza dal baricentro al bordo superiore del pacco
											END_IF
											
										RIBALTINO_DIRETTO:
										
											IF Forming^[WorkAreaState^[Mission^.PPlace].F].PackXP[WorkAreaState^[Mission^.PPlace].P].Grip = 0 THEN	// Aggiornamento altezza pallet con pacco in verticale (si considera la dimensione Y del pacco) 
												WorkArea^[Mission^.PPlace].H := WorkArea^[Mission^.PPlace].HPL +												// Altezza pallet + layers utilizzati
																	Forming^[WorkAreaState^[Mission^.PPlace].F].PackXP[WorkAreaState^[Mission^.PPlace].P].Z + 	// Quota "Z" del centro del pacco sulla piazzola, cioè altezza assoluta del baricentro
																	Mission^.XDim/2;													//Dimensione Y /2, indica la distanza dal baricentro al bordo superiore del pacco
											ELSIF Forming^[WorkAreaState^[cwa].F].PackXP[WorkAreaState^[cwa].P].Grip = 1 THEN
												WorkArea^[Mission^.PPlace].H := WorkArea^[Mission^.PPlace].HPL + 												// Altezza pallet + layers utilizzati
																	Forming^[WorkAreaState^[Mission^.PPlace].F].PackXP[WorkAreaState^[Mission^.PPlace].P].Z + 	// Quota "Z" del centro del pacco sulla piazzola, cioè altezza assoluta del baricentro
																	Mission^.ZDim/2;													//Dimensione Z /2, indica la distanza dal baricentro al bordo superiore del pacco
											END_IF
									END_CASE
								END_IF
								RestoreCWA^ := TRUE;
								PreviousPWA^ := pwa;
								WorkAreaManager^.State 	:= WAMANAGER_NOP;	// setto lo stato del WAMANAGER
								EXIT;
							ELSE																								// se dopo aver depositato un pacco, NON DEVO depositare NESSUNA falda
								(* Aggiorno Altezza Pallet su Ultimo Pacco *)
								IF Mission^.TPick = TPICK_PACK THEN													// Controllo che la missione  appena eseguita era un prelievo pacco ( dovrebbe sempre essere così!! mantenuto da vecchia gestione..)
									CASE TIPO_RIBALTINO OF
										RIBALTINO_DOPO_SQUADRO:
											IF Forming^[WorkAreaState^[Mission^.PPlace].F].PackXP[WorkAreaState^[Mission^.PPlace].P].Grip = 0 THEN	// Aggiornamento altezza pallet con pacco in verticale (si considera la dimensione Y del pacco) 
												WorkArea^[Mission^.PPlace].H := WorkArea^[Mission^.PPlace].HPL +												// Altezza pallet + layers utilizzati
																	Forming^[WorkAreaState^[Mission^.PPlace].F].PackXP[WorkAreaState^[Mission^.PPlace].P].Z + 	// Quota "Z" del centro del pacco sulla piazzola, cioè altezza assoluta del baricentro
																	Mission^.YDim/2;													//Dimensione Y /2, indica la distanza dal baricentro al bordo superiore del pacco
											ELSIF Forming^[WorkAreaState^[cwa].F].PackXP[WorkAreaState^[cwa].P].Grip = 1 THEN
												WorkArea^[Mission^.PPlace].H := WorkArea^[Mission^.PPlace].HPL + 												// Altezza pallet + layers utilizzati
																	Forming^[WorkAreaState^[Mission^.PPlace].F].PackXP[WorkAreaState^[Mission^.PPlace].P].Z + 	// Quota "Z" del centro del pacco sulla piazzola, cioè altezza assoluta del baricentro
																	Mission^.ZDim/2;													//Dimensione Z /2, indica la distanza dal baricentro al bordo superiore del pacco
											END_IF
											
										RIBALTINO_DIRETTO:
										
											IF Forming^[WorkAreaState^[Mission^.PPlace].F].PackXP[WorkAreaState^[Mission^.PPlace].P].Grip = 0 THEN	// Aggiornamento altezza pallet con pacco in verticale (si considera la dimensione Y del pacco) 
												WorkArea^[Mission^.PPlace].H := WorkArea^[Mission^.PPlace].HPL +												// Altezza pallet + layers utilizzati
																	Forming^[WorkAreaState^[Mission^.PPlace].F].PackXP[WorkAreaState^[Mission^.PPlace].P].Z + 	// Quota "Z" del centro del pacco sulla piazzola, cioè altezza assoluta del baricentro
																	Mission^.XDim/2;													//Dimensione Y /2, indica la distanza dal baricentro al bordo superiore del pacco
											ELSIF Forming^[WorkAreaState^[cwa].F].PackXP[WorkAreaState^[cwa].P].Grip = 1 THEN
												WorkArea^[Mission^.PPlace].H := WorkArea^[Mission^.PPlace].HPL + 												// Altezza pallet + layers utilizzati
																	Forming^[WorkAreaState^[Mission^.PPlace].F].PackXP[WorkAreaState^[Mission^.PPlace].P].Z + 	// Quota "Z" del centro del pacco sulla piazzola, cioè altezza assoluta del baricentro
																	Mission^.ZDim/2;													//Dimensione Z /2, indica la distanza dal baricentro al bordo superiore del pacco
											END_IF
									END_CASE
								END_IF
								(* Incremento WorkArea^[cwa].P (P=P+1) *)
								WorkAreaState^[Mission^.PPlace].P := WorkAreaState^[Mission^.PPlace].P + 1;
								(* Controllo Fine Pallettizzazione o Deposito Falda Dopo Strato Pacchi*)
								(* COME FACCIO A SAPERE SE è L'ULTIMO PACCO ? -> Si controlla la Grip=-1 *)
								(* Per sicurezza le controllo su entrambi le direzioni POSITIVA/NEGATIVA *)
								IF Forming^[WorkAreaState^[Mission^.PPlace].F].PackXP[WorkAreaState^[Mission^.PPlace].P].Grip = -1 OR
									Forming^[WorkAreaState^[Mission^.PPlace].F].PackXN[WorkAreaState^[Mission^.PPlace].P].Grip = -1 THEN
									IF NOT BypassTEST AND TRUE THEN //se true inizializza la piazzola a 1 pacco una volta completata la pallettizzazione
										WorkAreaState^[Mission^.PPlace].State := WORKAREA_STATE_OCCUPIED_WORKED;
										WorkAreaManager^.State 	:= WAMANAGER_NOP;	// setto lo stato del WAMANAGER
										RestoreCWA^ := TRUE;
										PreviousPWA^ := pwa;
										EXIT;
									ELSE
										WorkAreaState^[Mission^.PPlace].P := 1;
										WorkAreaManager^.State 	:= WAMANAGER_NOP;	// setto lo stato del WAMANAGER
										RestoreCWA^ := TRUE;
										PreviousPWA^ := pwa;
										EXIT;
									END_IF			
								END_IF
								WorkAreaManager^.State 	:= WAMANAGER_NOP;	// setto lo stato del WAMANAGER
								EXIT;
							END_IF								
					END_CASE	//riferito al case WorkAreaManager^.State
				ELSE			// riferito all' IF prima del  case WorkAreaManager^.State
					RestoreCWA^ := TRUE;
					PreviousPWA^ := pwa;
					WorkAreaState^[cwa].State := WORKAREA_STATE_OCCUPIED_DISABLED;
					EXIT;
				END_IF			// riferito all' IF prima del  case WorkAreaManager^.State

(**********************************************************************************************************************************************************************************)
(**********************************************************************************************************************************************************************************)
			(* ******************************************************************************************************** *)
						(* GESTIONE (Nastratura) o (Veicolo per prelievo/deposito PALLET FINITI/CATASTE/FALDE) *)
			(* ******************************************************************************************************** *)
(**********************************************************************************************************************************************************************************)
(**********************************************************************************************************************************************************************************)
			(* Occupied + Worked *)
			WORKAREA_STATE_OCCUPIED_WORKED:
				IF WorkArea^[cwa].Enable = 1 THEN
					IF NOT WorkArea^[cwa].RefuseLGV THEN		
						IF Forming^[WorkAreaState^[cwa].F].Tape = 0 THEN
							WorkAreaState^[cwa].State := WORKAREA_STATE_OCCUPIED_ENDED;
						ELSIF Forming^[WorkAreaState^[cwa].F].Tape = 1 THEN
							WorkAreaState^[cwa].State := WORKAREA_STATE_OCCUPIED_TAPING;
						END_IF
					ELSIF WorkArea^[cwa].RefuseLGV AND WorkArea^[cwa].LGV_Req = 1 THEN
						WorkArea^[cwa].LGV_Req := 0;
					END_IF	
				ELSE
					WorkAreaState^[cwa].State := WORKAREA_STATE_OCCUPIED_WORKED_DISABLED;
				END_IF
	
			(* Occupied + Worked + Disabled *)
			WORKAREA_STATE_OCCUPIED_WORKED_DISABLED:
				WorkArea^[cwa].LGV_Req := 0;
				IF WorkArea^[cwa].Enable = 1 THEN
					WorkAreaState^[cwa].State := WORKAREA_STATE_OCCUPIED_WORKED;
				ELSE
					;
				END_IF
	
			(* Occupied + Taping *)
			WORKAREA_STATE_OCCUPIED_TAPING:
				WorkArea^[cwa].LGV_Req := 0;
				IF WorkArea^[cwa].Enable = 1 THEN
					IF WorkArea^[cwa].LGV_Req = 0 AND  WorkArea^[cwa].LGV_ReqAbort THEN
						WorkAreaState^[cwa].State := WORKAREA_STATE_OCCUPIED_WORKING;
						WorkArea^[cwa].LGV_ReqAbort := FALSE;
					ELSE
						IF WorkArea^[cwa].Taped = 1 OR Forming^[WorkAreaState^[cwa].F].Tape = 0 THEN
							WorkAreaState^[cwa].State := WORKAREA_STATE_OCCUPIED_TAPED;
						END_IF
					END_IF	
				ELSE
					WorkAreaState^[cwa].State := WORKAREA_STATE_OCCUPIED_TAPING_DISABLED;
				END_IF
	
			(* Occupied + Taping + Disabled *)
			WORKAREA_STATE_OCCUPIED_TAPING_DISABLED:
				IF WorkArea^[cwa].Enable = 1 THEN
					WorkAreaState^[cwa].State := WORKAREA_STATE_OCCUPIED_TAPING;
				ELSE
					;
				END_IF
	
			(* Occupied + Taped *)
			WORKAREA_STATE_OCCUPIED_TAPED:
				IF WorkArea^[cwa].Enable = 1 THEN
					WorkAreaState^[cwa].State := WORKAREA_STATE_OCCUPIED_ENDED;
				ELSE
					WorkAreaState^[cwa].State := WORKAREA_STATE_OCCUPIED_TAPED_DISABLED;
				END_IF
	
			(* Occupied + Taped + Disabled *)
			WORKAREA_STATE_OCCUPIED_TAPED_DISABLED:
				WorkArea^[cwa].LGV_Req := 0;
				IF WorkArea^[cwa].Enable = 1 THEN
					WorkAreaState^[cwa].State := WORKAREA_STATE_OCCUPIED_TAPED;
				ELSE
					;
				END_IF
	
			(* Occupied + Ended *)
			WORKAREA_STATE_OCCUPIED_ENDED:
				IF WorkArea^[cwa].Enable = 1 THEN
					IF WorkArea^[cwa].Typology = TYPOLOGY_PALLET OR WorkArea^[cwa].Typology = TYPOLOGY_STACK AND NOT PX_WorkArea[cwa] THEN
						WorkAreaState^[cwa].State := WORKAREA_STATE_OCCUPIED_LGVREQ;
					END_IF	
				ELSE
					WorkAreaState^[cwa].State := WORKAREA_STATE_OCCUPIED_ENDED_DISABLED;
				END_IF
	
			(* Occupied + Ended + Disabled *)
			WORKAREA_STATE_OCCUPIED_ENDED_DISABLED:
				IF WorkArea^[cwa].Enable = 1 THEN
					WorkAreaState^[cwa].State := WORKAREA_STATE_OCCUPIED_ENDED;
				ELSE
					;
				END_IF
	
		 (* (* Occupied + LgvReq *)
			WORKAREA_STATE_OCCUPIED_LGVREQ:
				IF WorkArea^[cwa].Enable = 1 THEN
					; // Gestito dalla FB TFLGV
					IF WorkArea^[cwa].LGV_ReqAbort THEN
						WorkArea^[cwa].LGV_Req := 0;
						WorkArea^[cwa].LGV_ReqAbort := FALSE;
					ELSE
						WorkArea^[cwa].LGV_Req := 1; //aggiunto per comunicazione con LGV
						IF Forming^[WorkAreaState^[cwa].F].Tape = 1 AND WorkArea^[cwa].Taped < 1 THEN
							WorkArea^[cwa].LGV_Req := 0;
							WorkAreaState^[cwa].State := WORKAREA_STATE_OCCUPIED_WORKED;
						END_IF
					END_IF
				ELSE
					WorkAreaState^[cwa].State := WORKAREA_STATE_OCCUPIED_LGVREQ_DISABLED;				
				END_IF*)
				
			(* Occupied + LgvReq *)
			WORKAREA_STATE_OCCUPIED_LGVREQ:
				IF WorkArea^[cwa].Enable = 1 THEN
					IF Forming^[WorkAreaState^[cwa].F].Tape = 1 AND WorkArea^[cwa].Taped < 1 and WorkArea^[cwa].Typology = TYPOLOGY_PALLET THEN
						WorkArea^[cwa].LGV_Req := 0;
						WorkArea^[cwa].LGV_ReqAbort := FALSE;
						WorkAreaState^[cwa].State := WORKAREA_STATE_OCCUPIED_WORKED;
						EXIT;
					END_IF
					IF WorkArea^[cwa].LGV_ReqAbort THEN
						WorkArea^[cwa].LGV_Req := 0;
						WorkAreaState^[cwa].State := WORKAREA_STATE_OCCUPIED_LGVREQ_ABORT;
					ELSIF (NOT WorkArea^[cwa].LGV_ReqAbort AND WorkArea^[cwa].LGV_Req = 0) AND WorkArea^[cwa].Typology = TYPOLOGY_PALLET THEN
						IF Forming^[WorkAreaState^[cwa].F].PackXP[WorkAreaState^[cwa].P].Grip = -1 OR
							Forming^[WorkAreaState^[cwa].F].PackXN[WorkAreaState^[cwa].P].Grip = -1 THEN
							WorkArea^[cwa].LGV_Req := 1; 
						ELSE
							WorkAreaState^[cwa].State := WORKAREA_STATE_OCCUPIED_WORKING;
							EXIT;
						END_IF
					ELSE
						WorkArea^[cwa].LGV_Req := 1; 
					END_IF	
				ELSE
					WorkAreaState^[cwa].State := WORKAREA_STATE_OCCUPIED_LGVREQ_DISABLED;				
				END_IF
	
			(* Occupied + LgvReq + Disabled *)
			WORKAREA_STATE_OCCUPIED_LGVREQ_DISABLED:
				WorkArea^[cwa].LGV_Req := 0;
				IF WorkArea^[cwa].Enable = 1 THEN
					WorkAreaState^[cwa].State := WORKAREA_STATE_OCCUPIED_LGVREQ;
				ELSE
					;
				END_IF
				
			(* Occupied + LgvReqAbort *)
			WORKAREA_STATE_OCCUPIED_LGVREQ_ABORT:
				IF WorkArea^[cwa].Enable = 1 THEN
					IF (Forming^[WorkAreaState^[cwa].F].PackXP[WorkAreaState^[cwa].P].Grip <> -1 OR
						Forming^[WorkAreaState^[cwa].F].PackXN[WorkAreaState^[cwa].P].Grip <> -1) AND WorkArea^[cwa].LGV_ReqAbort THEN
							WorkAreaState^[cwa].State := WORKAREA_STATE_OCCUPIED_WORKING;
							WorkArea^[cwa].LGV_ReqAbort := FALSE;
							EXIT;
					ELSIF WorkArea^[cwa].LGV_ReqAbort THEN
						WorkArea^[cwa].LGV_Req := 0;
						//WorkArea^[cwa].LGV_ReqAbort := FALSE;
						EXIT;
					ELSIF WorkArea^[cwa].LGV_Req = 1 OR (Forming^[WorkAreaState^[cwa].F].PackXP[WorkAreaState^[cwa].P].Grip = -1 OR
						Forming^[WorkAreaState^[cwa].F].PackXN[WorkAreaState^[cwa].P].Grip = -1) THEN
							WorkAreaState^[cwa].State := WORKAREA_STATE_OCCUPIED_LGVREQ; 
							EXIT;
					END_IF
				ELSE
					;
				END_IF
	
			(* Occupied + LgvIn  - NOT USED !!!!!!!!!!!*)
			WORKAREA_STATE_OCCUPIED_LGVIN:
				IF WorkArea^[cwa].Enable = 1 THEN
					;
				ELSE
					;
				END_IF
	
			(* Occupied + LgvIn + Disabled  - NOT USED !!!!!!!!!!!*)
			WORKAREA_STATE_OCCUPIED_LGVIN_DISABLED:
				IF WorkArea^[cwa].Enable = 1 THEN
					;
				ELSE
					;
				END_IF
	
			(* Occupied + LgvEnd  - NOT USED !!!!!!!!!!!*)
			WORKAREA_STATE_OCCUPIED_LGVEND:
				IF WorkArea^[cwa].Enable = 1 THEN
					;
				ELSE
					;
				END_IF
	
			(* Occupied + LgvIn + Disabled - NOT USED !!!!!!!!!!! *)
			WORKAREA_STATE_OCCUPIED_LGVEND_DISABLED:
				IF WorkArea^[cwa].Enable = 1 THEN
					;
				ELSE
					;
				END_IF
	
			(* Error *)
			WORKAREA_STATE_ERROR:
				;
	
		ELSE		//riferito al WorkAreaState^[cwa].State								
			(* Stato Errato. viene Forzato lo stato di errore. Non dovrebbe MAI accadere *)
			WorkAreaState^[cwa].State := WORKAREA_STATE_ERROR;
				
		END_CASE;  //riferito al WorkAreaState^[cwa].State
	
	END_FOR			// riferito a FOR pwa:=1 TO MAXAREA DO


END_IF 				// riferito a IF WaitPositionRequest > 0 AND

//TFPalletizerWorkAreaManagerTF := TRUE;

END_FUNCTION_BLOCK

// ---- POUs/TFModules/Moduli TF/TFModulePalletizer_Ax.TcPOU
FUNCTION_BLOCK TFModulePalletizer_Ax
VAR_INPUT
	Cmd : CommandBuffer;
	Cfg : Config;
	IN : Module_Palletizer_Ax_IN;
	Ax : POINTER TO TFMotion;
	ManCmd : POINTER TO TFMachinePalletizer_AxeManCmd;
	AxisPar : POINTER TO Ax_Palletizer_Parameters;
	AxHomingParameters : POINTER TO AxHomingParameters;
	Programma : POINTER TO Descrittore_Programma;
	ProgrammaNEXT : POINTER TO Descrittore_Programma;
	AbilitaOffsetInUscitaTasteggio : BOOL := FALSE;	
	OffsetUscitaDaTasteggio: REAL := 0.0; 
	EncoderEsterno : POINTER TO GestioneEncoderEsterno;
	VelocitaDiUscitaDaTastatori : REAL;
	TempoRisalitaTastatori : REAL := 1;
	ByPassTastatoriInUscitaTasteggio : BOOL := FALSE;//Bypass sensore in uscita tastatori
	InterventoPxASpazio : BOOL := FALSE;
	SpazioInteventoPX : REAL := 20;
END_VAR
VAR_OUTPUT
	CmdExe : CommandExe;
	CmdExd : CommandExe;
	CmdNext : Command;
	CmdLog : CommandLog;
	ProgramLog : ProgrammaLog; 
	State : State;
	StateLog : StateLog;
	Error : Error;
	ErrorLog : ErrorLog;
	Warning : Warning;
	WarningLog : WarningLog;
	OUT : Module_Palletizer_Ax_OUT;
	//Status : TFTransportModuleStatus;
	QuotaAsseLetturaTasteggio : LREAL;
END_VAR
VAR
	Power : UINT;
	Init : BOOL;
	Timer : REAL;
	Timeout : REAL;
	TimerControlloCoppia : REAL;
	TempoFiltroTastatoriON : REAL;
	TempoFiltroTastatoriOFF : REAL;
	ParametersArray : ParametersArray;
	MAN_Actuator : UINT;
	MAN_Cmd : UINT;
	
	Px_Touch : BOOL;
	Px_TouchEmergency : BOOL;
	
	AggiornamentoParametriDone : BOOL;	  // va a true quando si carica un nuovo programma
	AggiornamentoLogProgrammiDone : BOOL := TRUE; // va a true quando è stato aggiornato il Log dei programmi eseguiti
	LancioNuovaMove	: BOOL; // Va a true quando dall'esterno viene lanciata una nuova move con un  nuovo programma.
	TempoControlloCoppia : REAL := 200;
	ContatoreNext : INT;
	ProgrammaLanciatoTrig : BOOL;
	ComandiMovimentoInviati : UINT;
	MovimentiDiretti : UINT;
	
	HomeDirect : BOOL;
	Spaziotastatori : Signal_SpaceFilter;
	PxSimulatoTasteggioSpazio: BOOL;
	DirezionePositivaRicercaTasteggio : BOOL;
END_VAR

IF NOT Init THEN
	TFCommandBufferClear(ADR(Cmd));
	TFCommandClear(ADR(CmdNext));
	TFCommandExeClear(ADR(CmdExe));
	TFStateUpdate(ADR(State),StateNOP);
	TFErrorClear(ADR(Error));
	TFWarningClear(ADR(Warning));
	Init := TRUE;
END_IF

(* Generic Timer - Add here all your Timers *)
TFTimerCall(ADR(Timer),Cfg.TimeBase);
TFTimerCall(ADR(Timeout),Cfg.TimeBase);
TFTimerCall(ADR(TimerControlloCoppia),Cfg.TimeBase);
TFTimerCall(ADR(TempoFiltroTastatoriON),Cfg.TimeBase);
TFTimerCall(ADR(TempoFiltroTastatoriOFF),Cfg.TimeBase);

IF Programma^.Torque > 0 THEN
	AxisPar^.MaxTorque	:= Programma^.Torque;
ELSE
	AxisPar^.MaxTorque	:= 50;
END_IF


(* Axis Call *)
Ax^();

Ax^.EnableTorqueCtrl := FALSE;
Ax^.EnableMoveAbsModifyContinuous := TRUE; //Abilitazione del move absoluto con cambi al volo

(* External To Buffered Command *)
TFCommandToNext(ADR(Cmd),ADR(CmdNext),ADR(CmdExe),ADR(Cfg),ADR(Error),ADR(ErrorLog),ADR(State));

(* Buffered To Exe Command *)
TFCommandToExecution(ADR(CmdNext),ADR(CmdExe),ADR(Error),ADR(ErrorLog),ADR(State),ADR(CmdLog));

(* Valorizzazione delle variabili utilizzando i parametri presenti nel programma da eseguire *)
(*IF CmdNext.Code = '' THEN
	IF Programma^.Stato = DA_ESEGUIRE THEN// AND NOT ProgrammaLanciatoTrig THEN
		AxisPar^.Acc 				:= Programma^.Accelerazione;
		AxisPar^.Dec 				:= Programma^.Decelerazione;
		AxisPar^.Vel 				:= Programma^.Velocita;
		AxisPar^.MaxTorque			:= Programma^.Torque;
		AxisPar^.Quota_Destinazione := Programma^.Quota_Destinazione;
		IF CmdExe.Code = CmdNOP THEN
			TFCommandSend(CmdMOVETOPOS,ParametersArray,Cmd);
			ComandiMovimentoInviati := ComandiMovimentoInviati+1;
		ELSIF CmdExe.Code = CmdMOVETOPOS THEN
			MovimentiDiretti := MovimentiDiretti +1;
		END_IF
		TFProgramLogUpdate(Programma,ADR(ProgramLog));
		//Programma^.Stato := IN_ESECUZIONE;
		ProgrammaLanciatoTrig := TRUE;
	END_IF
END_IF*)

(* Tastatori Pinza *)
//Px_Touch := IN.Px_Touch_1 AND IN.Px_Touch_2;
Px_Touch := IN.Px_Touch_1 OR IN.Px_Touch_2 OR In.Px_NuTouch;
Px_TouchEmergency := IN.Px_TouchEmergency_1 AND IN.Px_TouchEmergency_2;

Spaziotastatori(Sensor:= NOT Px_Touch,
						ActualPosition:=AX^.AxRef^.NcToPlc.ActPos,
						SpaceFilterON:=SpazioInteventoPX,
						SpaceFilterOFF:=SpazioInteventoPX,
						NegativeDirection := NOT Ax^.AxRef^.Status.PositiveDirection,
						AxisMoving:=Ax^.AxRef^.Status.Moving,
						EnableDirectStatusAxStop:=TRUE,
						SensorOUT=>PxSimulatoTasteggioSpazio);

IF CmdNext.Code = '' THEN
	IF Programma^.Stato = DA_ESEGUIRE THEN// AND NOT ProgrammaLanciatoTrig THEN
		AxisPar^.Acc 				:= Programma^.Accelerazione;
		AxisPar^.Dec 				:= Programma^.Decelerazione;
		AxisPar^.Vel 				:= Programma^.Velocita;
		AxisPar^.MaxTorque			:= Programma^.Torque;
		AxisPar^.Jerk				:= Programma^.Jerk;
		AxisPar^.Quota_Destinazione := Programma^.Quota_Destinazione;
		IF CmdExe.Code = CmdNOP THEN
			TFCommandSend(CmdMOVETOPOS,ParametersArray,Cmd);
			ComandiMovimentoInviati := ComandiMovimentoInviati+1;
		ELSIF CmdExe.Code = CmdMOVETOPOS THEN
			MovimentiDiretti := MovimentiDiretti +1;
		END_IF
		TFProgramLogUpdate(Programma,ADR(ProgramLog));
		ProgrammaLanciatoTrig := TRUE;
	ELSIF Programma^.Stato = IN_ESECUZIONE THEN
		IF AxisPar^.Acc <> Programma^.Accelerazione OR
		 AxisPar^.Dec 				<> Programma^.Decelerazione OR
		 AxisPar^.Vel 				<> Programma^.Velocita OR
		 AxisPar^.Jerk				<> Programma^.Jerk OR
		 AxisPar^.Quota_Destinazione <> Programma^.Quota_Destinazione THEN
			
			AxisPar^.Acc 				:= Programma^.Accelerazione;
			AxisPar^.Dec 				:= Programma^.Decelerazione;
			AxisPar^.Vel 				:= Programma^.Velocita;
			AxisPar^.MaxTorque			:= Programma^.Torque;
			AxisPar^.Jerk				:= Programma^.Jerk;
			AxisPar^.Quota_Destinazione := Programma^.Quota_Destinazione;
		END_IF
	
	END_IF
END_IF


IF CmdNext.Code <> '' THEN
	ContatoreNext := ContatoreNext +1;
END_IF

(* Exe Command *)
CASE CmdExe.Code OF

	(* ******************************************************************************************************** *)
	(* Nop  *)
	(* ******************************************************************************************************** *)
	CmdNOP:	;

	(* ******************************************************************************************************** *)
	(* Stop *)
	(* ******************************************************************************************************** *)
	CmdSTOP:
		CASE CmdExe.CmdCase OF
			
			(* Case 0 *)
			0: 	TFStateUpdate(ADR(State),StateSTOP_RUN);
				TFTimerSet(ADR(Timeout),2000,TRUE);
				TFCommandCase(ADR(CmdExe),1,CommandCase_INC);

			(* Case 1 - Clear All Commands*)
			1:	
				(* Se sto eseguendo un programma e mi arriva un comando di stop Imprevisto, setto lo stato del programma in interrotto *)
				IF Programma^.Stato = IN_ESECUZIONE THEN//AND Ax^.Command.MoveAbsolute THEN
					Programma^.Stato := INTERROTTO;
					//ProgrammaNEXT^.Stato := INTERROTTO;
					LancioNuovaMove := FALSE;
				END_IF
				ProgrammaLanciatoTrig := FALSE;
				AggiornamentoParametriDone := FALSE;			// Reset variabile per aggiornaento parametri asse
				AggiornamentoLogProgrammiDone := FALSE; 		// Reset variabile per aggiornaento Log dei Programmi
				Ax^.Command.ErrorReset 		:= FALSE;
				Ax^.Command.Home 			:= FALSE;
				Ax^.Command.MoveAbsolute 	:= FALSE;
				Ax^.Command.Halt 			:= FALSE;
				Ax^.Command.MoveJogNeg		:= FALSE;
				Ax^.Command.MoveJogPos		:= FALSE;
				Ax^.Command.HomeAbsEnc 		:= FALSE;
				TFCommandCase(ADR(CmdExe),1,CommandCase_INC);
				
			(* Case 2 *)
			2:	Ax^.Parameter.StopDeceleration 	:= AxisPar^.MaxDec;
				Ax^.Parameter.Deceleration 		:= AxisPar^.MaxDec;
				Ax^.Parameter.HaltDeceleration 	:= AxisPar^.MaxDec;
				Ax^.Parameter.Jerk				:= MaxJerk;
				Ax^.Command.Stop 				:= TRUE;
				IF Ax^.Status.StopDone THEN
					Ax^.Command.Stop := FALSE;
					TFCommandCase(ADR(CmdExe),100,CommandCase_JMP);
				ELSIF Ax^.Status.ErrorID <> ErrNULL THEN
					Ax^.Command.Stop := FALSE;
					TFError(ErrAXIS,Ax^.Status.ErrorID,ADR(CmdExe),ADR(State),ADR(Error),ADR(ErrorLog));
				ELSIF TFTimerDone(ADR(Timeout)) THEN
					Ax^.Command.Stop := FALSE;
					TFError(ErrTOSTOP,Ax^.Status.ErrorID,ADR(CmdExe),ADR(State),ADR(Error),ADR(ErrorLog));
				END_IF
			
			(* Case 100 *)
			100:TFStateUpdate(ADR(State),StateSTOP_END);
				TFCommandExeClear(ADR(CmdExe));

			ELSE
				TFError(ErrNOCMDCASE,ErrNULL,ADR(CmdExe),ADR(State),ADR(Error),ADR(ErrorLog));
		END_CASE
	
	(* ******************************************************************************************************** *)
	(* Error Reset *)
	(* ******************************************************************************************************** *)
	CmdRESET:
		CASE CmdExe.CmdCase OF

			(* Case 0 *)
			0: 	TFStateUpdate(ADR(State),StateRESET_RUN);
				TFTimerSet(ADR(Timeout),2000,TRUE);
				Ax^.Command.Home 			:= FALSE;
				Ax^.Command.MoveAbsolute 	:= FALSE;
				Ax^.Command.Halt 			:= FALSE;
				Ax^.Command.MoveJogNeg		:= FALSE;
				Ax^.Command.MoveJogPos		:= FALSE;
				Ax^.Command.HomeAbsEnc 		:= FALSE;
				IF NOT Ax^.Status.PowerActive AND Ax^.Status.ErrorID <> 0 THEN
					Ax^.Command.Power := FALSE;
				END_IF
				IF Programma^.Stato = IN_ESECUZIONE THEN//AND Ax^.Command.MoveAbsolute THEN
					Programma^.Stato := INTERROTTO;
					//ProgrammaNEXT^.Stato := INTERROTTO;
					LancioNuovaMove := FALSE;
				END_IF
				TFCommandCase(ADR(CmdExe),1,CommandCase_INC);
			
			(* Case 1 *)
			1:	Ax^.Command.ErrorReset := TRUE;
				AggiornamentoParametriDone := FALSE;
				ProgrammaLanciatoTrig := FALSE;				
				IF Ax^.Status.ErrorResetDone THEN
					Ax^.Command.ErrorReset := FALSE;
					IF Ax^.PowerEnable OR (Ax^.BrakeEnable AND Ax^.BrakePresent) THEN
						TFCommandCase(ADR(CmdExe),10,CommandCase_JMP);
					ELSE
						TFCommandCase(ADR(CmdExe),99,CommandCase_JMP);
					END_IF
				ELSIF TFTimerDone(ADR(Timeout)) THEN
					Ax^.Command.ErrorReset := FALSE;
					IF Ax^.Status.ErrorID <> ErrNULL THEN
						TFError(ErrAXIS,Ax^.Status.ErrorID,ADR(CmdExe),ADR(State),ADR(Error),ADR(ErrorLog));
					END_IF
					TFError(ErrTORESET,ErrNULL,ADR(CmdExe),ADR(State),ADR(Error),ADR(ErrorLog));
				END_IF

			(* Case 10 - Power On *)
			10:	
				Ax^.Command.Power := TRUE;
				
				IF Ax^.Status.PowerActive OR (Ax^.BrakeEnable AND Ax^.BrakePresent) THEN
					TFCommandCase(ADR(CmdExe),99,CommandCase_JMP);
				ELSIF Ax^.Status.ErrorID <> ErrNULL THEN
					Ax^.Command.Power := FALSE;
					TFError(ErrNOPOWER,Ax^.Status.ErrorID,ADR(CmdExe),ADR(State),ADR(Error),ADR(ErrorLog));
				ELSIF TFTimerDone(ADR(Timeout)) THEN
					Ax^.Command.Power := FALSE;
					TFError(ErrTOPOWERON,ErrNULL,ADR(CmdExe),ADR(State),ADR(Error),ADR(ErrorLog));
				END_IF
			
			(* Case 99 *)
			99:	TFErrorClear(ADR(Error));
				TFWarningClear(ADR(Warning));
				TFCommandCase(ADR(CmdExe),100,CommandCase_JMP);

			(* Case 100 *)
			100:TFStateUpdate(ADR(State),StateRESET_END);
				TFCommandExeClear(ADR(CmdExe));

			ELSE
				TFError(ErrNOCMDCASE,ErrNULL,ADR(CmdExe),ADR(State),ADR(Error),ADR(ErrorLog));
		END_CASE
	
	(* ******************************************************************************************************** *)
	(* Power *)
	(* ******************************************************************************************************** *)
	CmdPOWER:
		CASE CmdExe.CmdCase OF
			
			(* Case 0 *)
			0: 	TFStateUpdate(ADR(State),StatePOWER_RUN);
				TFTimerSet(ADR(Timeout),2500,TRUE);

				IF TFCommandParRead(CmdExe.Cmd.Parameter,ADR(ParametersArray),1) THEN
					Power := STRING_TO_UINT(ParametersArray.Parameters[0]);
				ELSE
					TFError(ErrCMDPARNUM,ErrNULL,ADR(CmdExe),ADR(State),ADR(Error),ADR(ErrorLog));
					RETURN;
				END_IF

				IF Power = 1 THEN
					TFCommandCase(ADR(CmdExe),5,CommandCase_JMP);
				ELSE
					TFCommandCase(ADR(CmdExe),20,CommandCase_JMP);
				END_IF
				
			5:
				Ax^.Command.ErrorReset := TRUE;
				AggiornamentoParametriDone := FALSE;
				ProgrammaLanciatoTrig := FALSE;				
				IF Ax^.Status.ErrorResetDone THEN
					Ax^.Command.ErrorReset := FALSE;
					TFCommandCase(ADR(CmdExe),10,CommandCase_JMP);
				ELSIF TFTimerDone(ADR(Timeout)) THEN
					Ax^.Command.ErrorReset := FALSE;
					IF Ax^.Status.ErrorID <> ErrNULL THEN
						TFError(ErrAXIS,Ax^.Status.ErrorID,ADR(CmdExe),ADR(State),ADR(Error),ADR(ErrorLog));
					END_IF
					TFError(ErrTORESET,ErrNULL,ADR(CmdExe),ADR(State),ADR(Error),ADR(ErrorLog));
				END_IF	
				
			(* Case 10 - Power On *)
			10:	Ax^.Command.Power := TRUE;
				
				IF Ax^.Status.PowerActive OR (Ax^.BrakeEnable AND Ax^.BrakePresent) THEN
					TFCommandCase(ADR(CmdExe),100,CommandCase_JMP);
				ELSIF Ax^.Status.ErrorID <> ErrNULL THEN
					Ax^.Command.Power := FALSE;
					TFError(ErrNOPOWER,Ax^.Status.ErrorID,ADR(CmdExe),ADR(State),ADR(Error),ADR(ErrorLog));
				ELSIF TFTimerDone(ADR(Timeout)) THEN
					Ax^.Command.Power := FALSE;
					TFError(ErrTOPOWERON,ErrNULL,ADR(CmdExe),ADR(State),ADR(Error),ADR(ErrorLog));
				END_IF
			
			(* Case 20 - Power Off *)
			20:	Ax^.Command.Power := FALSE;
				
				IF NOT Ax^.Status.PowerActive THEN
					TFCommandCase(ADR(CmdExe),100,CommandCase_JMP);
				ELSIF Ax^.Status.ErrorID <> ErrNULL THEN
					TFError(ErrAXIS,Ax^.Status.ErrorID,ADR(CmdExe),ADR(State),ADR(Error),ADR(ErrorLog));
				ELSIF TFTimerDone(ADR(Timeout)) THEN
					TFError(ErrTOPOWEROFF,ErrNULL,ADR(CmdExe),ADR(State),ADR(Error),ADR(ErrorLog));
				END_IF
				
			(* Case 100 *)
			100:TFStateUpdate(ADR(State),StatePOWER_END);
				TFCommandExeClear(ADR(CmdExe));

			ELSE
				TFError(ErrNOCMDCASE,ErrNULL,ADR(CmdExe),ADR(State),ADR(Error),ADR(ErrorLog));
		END_CASE
	
	(* ******************************************************************************************************** *)
	(* Home *)
	(* ******************************************************************************************************** *)
	CmdHOME:
		CASE CmdExe.CmdCase OF

			(* Case 0 *)
			0: 	TFStateUpdate(ADR(State),StateHOME_RUN);
				TFTimerSet(ADR(Timeout),120000,TRUE);
				
				IF TFCommandParRead(CmdExe.Cmd.Parameter,ADR(ParametersArray),1) THEN
					HomeDirect := STRING_TO_BOOL(ParametersArray.Parameters[0]);				
				ELSE
					TFError(ErrCMDPARNUM,ErrNULL,ADR(CmdExe),ADR(State),ADR(Error),ADR(ErrorLog));
					RETURN;
				END_IF
				(* Valuto se devo fare l'home direct *)
				IF HomeDirect THEN
					IF AxHomingParameters^.TipoHoming = HOMING_STANDARD THEN
						TFCommandCase(ADR(CmdExe),89,CommandCase_JMP);
					ELSIF  AxHomingParameters^.TipoHoming = HOMING_ASSE_PINZA THEN
						TFCommandCase(ADR(CmdExe),62,CommandCase_JMP);
					END_IF
				ELSE
					TFCommandCase(ADR(CmdExe),1,CommandCase_INC);
				END_IF
				
				
			(* Case 1 - Stop Asse *)
			1:	Ax^.Command.Stop := TRUE;
				IF Ax^.Status.StopDone THEN
					Ax^.Command.Stop := FALSE;
					TFCommandCase(ADR(CmdExe),1,CommandCase_INC);
				ELSIF TFTimerDone(ADR(Timeout)) THEN
					Ax^.Command.Stop := FALSE;
					TFError(ErrTOHOME,ErrNULL,ADR(CmdExe),ADR(State),ADR(Error),ADR(ErrorLog));
				END_IF

			(* Case 2 - Power ON Asse *)
			2:	CASE Ax^.EncoderType OF
					INCREMENTAL_ENCODER:
						Ax^.Command.Power := TRUE;
						IF Ax^.Status.PowerActive THEN
							TFTimerSet(ADR(Timeout),120000,TRUE);
						ELSIF Ax^.Status.ErrorID <> ErrNULL THEN
							Ax^.Command.Power := FALSE;
							TFError(ErrAXIS,Ax^.Status.ErrorID,ADR(CmdExe),ADR(State),ADR(Error),ADR(ErrorLog));
						ELSIF TFTimerDone(ADR(Timeout)) THEN
							Ax^.Command.Power := FALSE;
							TFError(ErrTOHOME,ErrNULL,ADR(CmdExe),ADR(State),ADR(Error),ADR(ErrorLog));
						END_IF
						TFCommandCase(ADR(CmdExe),1,CommandCase_INC);
					ABSOLUTE_ENCODER:
						IF AxHomingParameters^.TipoHoming = HOMING_STANDARD THEN
							TFCommandCase(ADR(CmdExe),6,CommandCase_JMP);
						ELSIF  AxHomingParameters^.TipoHoming = HOMING_ASSE_PINZA THEN
							TFCommandCase(ADR(CmdExe),62,CommandCase_JMP);
						END_IF	
				ELSE
					TFCommandCase(ADR(CmdExe),100,CommandCase_JMP);
				END_CASE
				
			(* Case 3 - Gestione encoder Relativo *)
			3:	Ax^.Command.Home := TRUE;
				Ax^.Parameter.HomePosition  := AxisPar^.HomeDefine;
				Ax^.Parameter.HomeMode 		:= HomeModeDefault;
				Ax^.Parameter.Torque		:= 50;
				Ax^.Parameter.TorqueMax		:= 100;
				IF Ax^.Status.HomeDone THEN
					Ax^.Command.Home := FALSE;
					TFTimerSet(ADR(Timeout),120000,TRUE);
					TFCommandCase(ADR(CmdExe),100,CommandCase_JMP);
				ELSIF Ax^.Status.ErrorID <> ErrNULL THEN
					Ax^.Command.Home := FALSE;
					TFError(ErrAXIS,Ax^.Status.ErrorID,ADR(CmdExe),ADR(State),ADR(Error),ADR(ErrorLog));
				ELSIF TFTimerDone(ADR(Timeout)) THEN
					Ax^.Command.Home := FALSE;
					TFError(ErrTOHOME,ErrNULL,ADR(CmdExe),ADR(State),ADR(Error),ADR(ErrorLog));
				ELSIF IN.Enable_TouchEmergency^ AND (NOT Px_TouchEmergency) THEN
					Ax^.Command.Home := FALSE;
					TFError(ErrTOUCHEMERGENCY,ErrNULL,ADR(CmdExe),ADR(State),ADR(Error),ADR(ErrorLog));
					RegistroAlarma2205 := 21 ;
				END_IF	
			
			(* Case 4 - Mi porto in posizione di Home *)
			4:	Ax^.Command.MoveAbsolute := TRUE;
				Ax^.Parameter.Position 		:= AxisPar^.HomePosition;
				Ax^.Parameter.Acceleration 	:= AxisPar^.JOGAcc;
				Ax^.Parameter.Deceleration 	:= AxisPar^.JOGDec;
				Ax^.Parameter.Jerk 			:= AxisPar^.Jerk;
				Ax^.Parameter.Torque		:= 50;
				Ax^.Parameter.TorqueMax		:= 100;
				Ax^.Parameter.Velocity := AxisPar^.MaxVel * 0.1 ;

				IF Ax^.Status.MoveAbsoluteDone THEN
					Ax^.Command.MoveAbsolute := FALSE;
					TFCommandCase(ADR(CmdExe),100,CommandCase_JMP);
				ELSIF Ax^.Status.ErrorID <> ErrNULL THEN
					Ax^.Command.Home := FALSE;
					TFError(ErrAXIS,Ax^.Status.ErrorID,ADR(CmdExe),ADR(State),ADR(Error),ADR(ErrorLog));
				ELSIF TFTimerDone(ADR(Timeout)) THEN
					Ax^.Command.Home := FALSE;
					TFError(ErrTOHOME,ErrNULL,ADR(CmdExe),ADR(State),ADR(Error),ADR(ErrorLog));
				ELSIF IN.Enable_TouchEmergency^ AND (NOT Px_TouchEmergency) THEN
					Ax^.Command.MoveAbsolute := FALSE;
					TFError(ErrTOUCHEMERGENCY,ErrNULL,ADR(CmdExe),ADR(State),ADR(Error),ADR(ErrorLog));
					RegistroAlarma2205 := 22 ;
				END_IF
			
			(* Case 6 - Gestione encoder ASSOLUTO *)
			6:	Ax^.Command.Home := TRUE;
				Ax^.Parameter.HomePosition  := LREAL_TO_REAL(Ax^.AxRef^.NcToPlc.ActPos);
				Ax^.Parameter.HomeMode 		:= HomeModeDirect;
				Ax^.Parameter.Torque		:= 50;
				Ax^.Parameter.TorqueMax		:= 100;
				IF Ax^.Status.HomeDone THEN
					Ax^.Command.Home := FALSE;
					TFTimerSet(ADR(Timeout),120000,TRUE);
					TFCommandCase(ADR(CmdExe),1,CommandCase_INC);
				ELSIF Ax^.Status.ErrorID <> ErrNULL THEN
					Ax^.Command.Home := FALSE;
					TFError(ErrAXIS,Ax^.Status.ErrorID,ADR(CmdExe),ADR(State),ADR(Error),ADR(ErrorLog));
				ELSIF TFTimerDone(ADR(Timeout)) THEN
					Ax^.Command.Home := FALSE;
					TFError(ErrTOHOME,ErrNULL,ADR(CmdExe),ADR(State),ADR(Error),ADR(ErrorLog));
				ELSIF IN.Enable_TouchEmergency^ AND (NOT Px_TouchEmergency) THEN
					Ax^.Command.Home := FALSE;
					TFError(ErrTOUCHEMERGENCY,ErrNULL,ADR(CmdExe),ADR(State),ADR(Error),ADR(ErrorLog));
					RegistroAlarma2205 := 23 ;
				END_IF	
			
			(* Case 7 - Mi porto in posizione di Home *)
			7:	Ax^.Command.MoveAbsolute := TRUE;
				Ax^.Parameter.Position 		:= AxisPar^.HomePosition;
				Ax^.Parameter.Acceleration 	:= AxisPar^.JOGAcc;
				Ax^.Parameter.Deceleration 	:= AxisPar^.JOGDec;
				Ax^.Parameter.Jerk 			:= AxisPar^.Jerk;
				Ax^.Parameter.Torque		:= 50;
				Ax^.Parameter.TorqueMax		:= 100;
				Ax^.Parameter.Velocity 		:= AxisPar^.MaxVel * 0.1 ;

				IF Ax^.Status.MoveAbsoluteDone THEN
					Ax^.Command.MoveAbsolute := FALSE;
					TFCommandCase(ADR(CmdExe),100,CommandCase_JMP);
				ELSIF Ax^.Status.ErrorID <> ErrNULL THEN
					Ax^.Command.Home := FALSE;
					TFError(ErrAXIS,Ax^.Status.ErrorID,ADR(CmdExe),ADR(State),ADR(Error),ADR(ErrorLog));
				ELSIF TFTimerDone(ADR(Timeout)) THEN
					Ax^.Command.Home := FALSE;
					TFError(ErrTOHOME,ErrNULL,ADR(CmdExe),ADR(State),ADR(Error),ADR(ErrorLog));
				ELSIF IN.Enable_TouchEmergency^ AND (NOT Px_TouchEmergency) THEN
					Ax^.Command.MoveAbsolute := FALSE;
					TFError(ErrTOUCHEMERGENCY,ErrNULL,ADR(CmdExe),ADR(State),ADR(Error),ADR(ErrorLog));
					RegistroAlarma2205 := 24 ;
				END_IF
				
			(* Jog fino alla lettura del sensore *)
			60:
				Ax^.Parameter.Torque		:= AxisPar^.MaxTorque;
				Ax^.Parameter.TorqueMax		:= 100;
				Ax^.Parameter.Acceleration 	:= AxisPar^.JOGAcc;
				Ax^.Parameter.Deceleration 	:= AxisPar^.JOGDec;
				Ax^.Parameter.Jerk 			:= AxisPar^.Jerk;
				Ax^.Parameter.JogVelocity 	:= AxisPar^.ManSlowVel / 100.0 * AxisPar^.MaxVel;
				IF AxHomingParameters^.InvertiDirezione THEN
					Ax^.Command.MoveJogPos := TRUE;
				ELSE
					Ax^.Command.MoveJogNeg := TRUE;
				END_IF
				IF Ax^.PxHome THEN
					Ax^.Command.MoveJogPos := FALSE;
					Ax^.Command.MoveJogNeg := FALSE;
					TFCommandCase(ADR(CmdExe),1,CommandCase_INC);
				END_IF
				IF Ax^.Status.ErrorID <> ErrNULL THEN
					Ax^.Command.MoveJogNeg  := FALSE;
					Ax^.Command.MoveJogPos := FALSE;
					TFError(ErrAXIS,Ax^.Status.ErrorID,ADR(CmdExe),ADR(State),ADR(Error),ADR(ErrorLog));
				ELSIF TFTimerDone(ADR(Timeout)) THEN
					Ax^.Command.MoveJogNeg  := FALSE;
					Ax^.Command.MoveJogPos := FALSE;
					TFError(ErrTOHOME,ErrNULL,ADR(CmdExe),ADR(State),ADR(Error),ADR(ErrorLog));
				ELSIF IN.Enable_TouchEmergency^ AND (NOT Px_TouchEmergency) THEN
					Ax^.Command.MoveJogNeg  := FALSE;
					Ax^.Command.MoveJogPos := FALSE;
					TFError(ErrTOUCHEMERGENCY,ErrNULL,ADR(CmdExe),ADR(State),ADR(Error),ADR(ErrorLog));
					RegistroAlarma2205 := 25 ;
				END_IF
				
			(* Jog fino a liberare il sensore *)	
			61:
				Ax^.Parameter.Torque		:= AxisPar^.MaxTorque;
				Ax^.Parameter.TorqueMax		:= 100;
				Ax^.Parameter.Acceleration 	:= AxisPar^.JOGAcc;
				Ax^.Parameter.Deceleration 	:= AxisPar^.JOGDec;
				Ax^.Parameter.Jerk 			:= AxisPar^.Jerk;
				Ax^.Parameter.JogVelocity 	:=  5/100.0 * AxisPar^.MaxVel;
				IF AxHomingParameters^.InvertiDirezione THEN
					Ax^.Command.MoveJogNeg := TRUE;
				ELSE
					Ax^.Command.MoveJogPos := TRUE;
				END_IF
				IF NOT Ax^.PxHome THEN
					Ax^.Command.MoveJogNEG := FALSE;
					TFCommandCase(ADR(CmdExe),1,CommandCase_INC);
				END_IF
				IF Ax^.Status.ErrorID <> ErrNULL THEN
					Ax^.Command.MoveJogNeg  := FALSE;
					Ax^.Command.MoveJogPos := FALSE;
					TFError(ErrAXIS,Ax^.Status.ErrorID,ADR(CmdExe),ADR(State),ADR(Error),ADR(ErrorLog));
				ELSIF TFTimerDone(ADR(Timeout)) THEN
					Ax^.Command.MoveJogNeg  := FALSE;
					Ax^.Command.MoveJogPos := FALSE;
					TFError(ErrTOHOME,ErrNULL,ADR(CmdExe),ADR(State),ADR(Error),ADR(ErrorLog));
				ELSIF IN.Enable_TouchEmergency^ AND (NOT Px_TouchEmergency) THEN
					Ax^.Command.MoveJogNeg  := FALSE;
					Ax^.Command.MoveJogPos := FALSE;
					TFError(ErrTOUCHEMERGENCY,ErrNULL,ADR(CmdExe),ADR(State),ADR(Error),ADR(ErrorLog));
					RegistroAlarma2205 := 26 ;
				END_IF
				
			(* Eseguo Homing *)	
			62:
				(*Ax^.Command.HomeAbsEnc := TRUE;
				Ax^.Parameter.HomePosition  := AxisPar^.HomeDefine;
				Ax^.Parameter.Torque		:= 50;
				Ax^.Parameter.TorqueMax		:= 100;
				IF Ax^.Status.HomeAbsEncDone THEN
					Ax^.Command.HomeAbsEnc := FALSE;
					TFTimerSet(ADR(Timeout),120000,TRUE);
					TFCommandCase(ADR(CmdExe),100,CommandCase_JMP);
				ELSIF Ax^.Status.ErrorID <> ErrNULL THEN
					Ax^.Command.HomeAbsEnc := FALSE;
					TFError(ErrAXIS,Ax^.Status.ErrorID,ADR(CmdExe),ADR(State),ADR(Error),ADR(ErrorLog));
				ELSIF TFTimerDone(ADR(Timeout)) THEN
					Ax^.Command.HomeAbsEnc := FALSE;
					TFError(ErrTOHOME,ErrNULL,ADR(CmdExe),ADR(State),ADR(Error),ADR(ErrorLog));
				ELSIF IN.Enable_TouchEmergency^ AND (NOT Px_TouchEmergency) THEN
					Ax^.Command.HomeAbsEnc := FALSE;
					TFError(ErrTOUCHEMERGENCY,ErrNULL,ADR(CmdExe),ADR(State),ADR(Error),ADR(ErrorLog));
				END_IF*)
				Ax^.Parameter.HomeVelocity  := AxisPar^.HomeVelocity;
				Ax^.Command.HomeAbsEnc 		:= TRUE;
				Ax^.Parameter.HomePosition  := AxisPar^.HomeDefine;
				Ax^.Parameter.HomeInvertDirection  := AxHomingParameters^.InvertiDirezione;
				Ax^.Parameter.Torque		:= 50;
				Ax^.Parameter.TorqueMax		:= 100;
				IF Ax^.Status.HomeAbsEncDone THEN
					Ax^.Command.HomeAbsEnc := FALSE;
					TFTimerSet(ADR(Timeout),120000,TRUE);
					TFCommandCase(ADR(CmdExe),100,CommandCase_JMP);
				ELSIF IN.Enable_TouchEmergency^ AND (NOT Px_TouchEmergency) THEN  
					Ax^.Command.MoveJogPos := FALSE;
					Ax^.Command.MoveJogNeg := FALSE;
					Ax^.Command.HomeAbsEnc := FALSE;
					TFError(ErrTOUCHEMERGENCY,ErrNULL,ADR(CmdExe),ADR(State),ADR(Error),ADR(ErrorLog));
					RegistroAlarma2205 := 27 ;
				ELSIF Ax^.Status.ErrorID <> ErrNULL THEN
					Ax^.Command.MoveJogPos := FALSE;
					Ax^.Command.MoveJogNeg := FALSE;
					Ax^.Command.HomeAbsEnc := FALSE;
					TFError(ErrAXIS,Ax^.Status.ErrorID,ADR(CmdExe),ADR(State),ADR(Error),ADR(ErrorLog));
				ELSIF TFTimerDone(ADR(Timeout))THEN
					Ax^.Command.MoveJogPos := FALSE;
					Ax^.Command.MoveJogNeg := FALSE;
					Ax^.Command.HomeAbsEnc := FALSE;
					TFError(ErrTOHOME,ErrNULL,ADR(CmdExe),ADR(State),ADR(Error),ADR(ErrorLog));
				END_IF
			
			(* Case 89 - HomeDirect *)
			89:	Ax^.Command.Home 			:= TRUE;
				Ax^.Parameter.HomePosition  := LREAL_TO_REAL(Ax^.AxRef^.NcToPlc.ActPos);
				Ax^.Parameter.HomeMode 		:= HomeModeDirect;
				Ax^.Parameter.Torque		:= 50;
				Ax^.Parameter.TorqueMax		:= 100;
				IF Ax^.Status.HomeDone THEN
					Ax^.Command.Home := FALSE;
					TFTimerSet(ADR(Timeout),120000,TRUE);
					TFCommandCase(ADR(CmdExe),100,CommandCase_JMP);
				ELSIF Ax^.Status.ErrorID <> ErrNULL THEN
					Ax^.Command.Home := FALSE;
					TFError(ErrAXIS,Ax^.Status.ErrorID,ADR(CmdExe),ADR(State),ADR(Error),ADR(ErrorLog));
				ELSIF TFTimerDone(ADR(Timeout)) THEN
					Ax^.Command.Home := FALSE;
					TFError(ErrTOHOME,ErrNULL,ADR(CmdExe),ADR(State),ADR(Error),ADR(ErrorLog));
				ELSIF IN.Enable_TouchEmergency^ AND (NOT Px_TouchEmergency) THEN
					Ax^.Command.Home := FALSE;
					TFError(ErrTOUCHEMERGENCY,ErrNULL,ADR(CmdExe),ADR(State),ADR(Error),ADR(ErrorLog));
					RegistroAlarma2205 := 28 ;
				END_IF
	
			(* Case 90 - Mi porto in posizione di Home *)
			90:	Ax^.Command.MoveAbsolute := TRUE;
				Ax^.Parameter.Position 		:= AxisPar^.HomePosition;
				Ax^.Parameter.Acceleration 	:= AxisPar^.JOGAcc;
				Ax^.Parameter.Deceleration 	:= AxisPar^.JOGDec;
				Ax^.Parameter.Jerk 			:= AxisPar^.Jerk;
				Ax^.Parameter.Torque		:= 50;
				Ax^.Parameter.TorqueMax		:= 100;
				Ax^.Parameter.Velocity 		:= AxisPar^.MaxVel * 0.1 ;

				IF Ax^.Status.MoveAbsoluteDone THEN
					Ax^.Command.MoveAbsolute := FALSE;
					TFCommandCase(ADR(CmdExe),100,CommandCase_JMP);
				ELSIF Ax^.Status.ErrorID <> ErrNULL THEN
					Ax^.Command.Home := FALSE;
					TFError(ErrAXIS,Ax^.Status.ErrorID,ADR(CmdExe),ADR(State),ADR(Error),ADR(ErrorLog));
				ELSIF TFTimerDone(ADR(Timeout)) THEN
					Ax^.Command.Home := FALSE;
					TFError(ErrTOHOME,ErrNULL,ADR(CmdExe),ADR(State),ADR(Error),ADR(ErrorLog));
				ELSIF IN.Enable_TouchEmergency^ AND (NOT Px_TouchEmergency) THEN
					Ax^.Command.MoveAbsolute := FALSE;
					TFError(ErrTOUCHEMERGENCY,ErrNULL,ADR(CmdExe),ADR(State),ADR(Error),ADR(ErrorLog));
					RegistroAlarma2205 := 29 ;
				END_IF
				
			(* Case 100 *)
			100:TFStateUpdate(ADR(State),StateHOME_END);
				HomeDirect:=FALSE;
				TFCommandExeClear(ADR(CmdExe));

			ELSE
				TFError(ErrNOCMDCASE,ErrNULL,ADR(CmdExe),ADR(State),ADR(Error),ADR(ErrorLog));
		END_CASE

	(* ******************************************************************************************************** *)
	(* Manual *)
	(* ******************************************************************************************************** *)
	CmdMAN:
		CASE CmdExe.CmdCase OF
			(* Case 0 *)
			0: 	TFStateUpdate(ADR(State),StateMAN_RUN);
				TFTimerSet(ADR(Timeout),10,TRUE);
				IF TFCommandParRead(CmdExe.Cmd.Parameter,ADR(ParametersArray),2) THEN
					MAN_Actuator	:= STRING_TO_UINT(ParametersArray.Parameters[0]);
					MAN_Cmd		:= STRING_TO_UINT(ParametersArray.Parameters[1]);
					IF ManCmd^.JogFast THEN
						Ax^.Parameter.JogVelocity := AxisPar^.ManFastVel / 100.0 * AxisPar^.MaxVel;
					ELSE
						Ax^.Parameter.JogVelocity := AxisPar^.ManSlowVel / 100.0 * AxisPar^.MaxVel;
					END_IF
				ELSE
					TFError(ErrCMDPARNUM,ErrNULL,ADR(CmdExe),ADR(State),ADR(Error),ADR(ErrorLog));
					RETURN;
				END_IF;

				CASE MAN_Actuator OF
					(* Case 0..99 for Actuators *)
					(* Case 100..199  for Axis *)

					(* Case Nop *)
					0:	;

					(* Case 1: *)
					1:	CASE MAN_Cmd OF
							0:	;

							ELSE
								TFError(ErrNOCMDCASE,ErrNULL,ADR(CmdExe),ADR(State),ADR(Error),ADR(ErrorLog));
						END_CASE;

					100:CASE MAN_Cmd OF
							0:	;

							(* Case 10: *)
							10:	;
								
							(* Case 11: Jog + *)
							11:	
								Ax^.Parameter.Torque		:= 100;//AxisPar^.MaxTorque;
								Ax^.Parameter.TorqueMax		:= 100;
								Ax^.Parameter.Acceleration 	:= AxisPar^.JOGAcc;
								Ax^.Parameter.Deceleration 	:= AxisPar^.JOGDec;
								Ax^.Parameter.Jerk 			:= AxisPar^.Jerk;
								IF Ax^.Status.ActPosition >= AxisPar^.MaxPosition AND IN.Enable_TouchEmergency^ THEN
									Ax^.Command.MoveJogPos := FALSE;
								ELSE
									Ax^.Command.MoveJogPos := TRUE;
								END_IF
								IF IN.Enable_TouchEmergency^ AND (NOT Px_TouchEmergency) THEN
									Ax^.Command.MoveJogPos := FALSE;
									TFError(ErrTOUCHEMERGENCY,ErrNULL,ADR(CmdExe),ADR(State),ADR(Error),ADR(ErrorLog));
									RegistroAlarma2205 := 30 ;
								END_IF			
								
							(* Case 12: Jog - *)
							12:	IF Ax^.Status.ActPosition <= AxisPar^.MinPosition AND IN.Enable_TouchEmergency^ THEN
									Ax^.Command.MoveJogNeg := FALSE;
								ELSE
									Ax^.Command.MoveJogNeg := TRUE;
								END_IF
								Ax^.Parameter.Torque		:= 100;//AxisPar^.MaxTorque;
								Ax^.Parameter.TorqueMax		:= 100;
								Ax^.Parameter.Acceleration 	:= AxisPar^.JOGAcc;
								Ax^.Parameter.Deceleration 	:= AxisPar^.JOGDec;
								Ax^.Parameter.Jerk 			:= AxisPar^.Jerk;
								//IF ManCmd^.JogFast THEN
								//	Ax^.Parameter.JogVelocity := AxisPar^.ManFastVel / 100.0 * AxisPar^.MaxVel;
								//ELSE
								//	Ax^.Parameter.JogVelocity := AxisPar^.ManSlowVel / 100.0 * AxisPar^.MaxVel;
								//END_IF
								IF IN.Enable_TouchEmergency^ AND (NOT Px_TouchEmergency) THEN
									Ax^.Command.MoveJogNEG := FALSE;
									TFError(ErrTOUCHEMERGENCY,ErrNULL,ADR(CmdExe),ADR(State),ADR(Error),ADR(ErrorLog));
									RegistroAlarma2205 := 31 ;
								END_IF	
							
							(* Case 13 - Move Absolute a posizione data *)
							13:
								TFTimerSet(ADR(Timeout),30000,TRUE);	
								Ax^.Command.MoveAbsolute 	:= TRUE;
								Ax^.Parameter.Position 		:= LREAL_TO_REAL(AxisPar^.Quota_Destinazione);
								Ax^.Parameter.Acceleration 	:= AxisPar^.JOGAcc;
								Ax^.Parameter.Deceleration 	:= AxisPar^.JOGDec;
								Ax^.Parameter.Jerk 			:= AxisPar^.Jerk;
								Ax^.Parameter.Torque		:= 50;
								Ax^.Parameter.TorqueMax		:= 100;
								Ax^.Parameter.Velocity := AxisPar^.MaxVel * 0.1 ;
								TFCommandCase(ADR(CmdExe),13,CommandCase_JMP);
								
							(* Esecuzione Homing Asse*)
							20: TFTimerSet(ADR(Timeout),120000,TRUE);
								CASE Ax^.EncoderType OF
									INCREMENTAL_ENCODER:
										TFCommandCase(ADR(CmdExe),20,CommandCase_JMP);
									ABSOLUTE_ENCODER:
										IF AxHomingParameters^.TipoHoming = HOMING_STANDARD THEN
											TFCommandCase(ADR(CmdExe),30,CommandCase_JMP);
										ELSIF AxHomingParameters^.TipoHoming = HOMING_ASSE_PINZA THEN
											TFCommandCase(ADR(CmdExe),30,CommandCase_JMP);
										END_IF	
								ELSE
									TFCommandCase(ADR(CmdExe),100,CommandCase_JMP);
								END_CASE
	
						ELSE
							TFError(ErrNOCMDCASE,ErrNULL,ADR(CmdExe),ADR(State),ADR(Error),ADR(ErrorLog));
						END_CASE;

					ELSE
						TFError(ErrNOCMDCASE,ErrNULL,ADR(CmdExe),ADR(State),ADR(Error),ADR(ErrorLog));
				END_CASE
				IF CmdExe.CmdCase = 0 THEN
					TFCommandCase(ADR(CmdExe),1,CommandCase_INC);
				END_IF

			(* Case 1 *)
			1: 	IF (MAN_Cmd = 0) OR TFTimerDone(ADR(Timeout)) THEN
					(* Clear All Output Here *)
					Ax^.Command.Home := FALSE;
					Ax^.Command.MoveJogPos := FALSE;
					Ax^.Command.MoveJogNeg := FALSE;
					
					TFStateUpdate(ADR(State),StateMAN_END);
					TFCommandExeClear(ADR(CmdExe));
				END_IF
				IF IN.Enable_TouchEmergency^ AND (NOT Px_TouchEmergency) THEN
					Ax^.Command.Home := FALSE;
					Ax^.Command.MoveJogPos := FALSE;
					Ax^.Command.MoveJogNeg := FALSE;
					TFCommandExeClear(ADR(CmdExe));
					TFError(ErrTOUCHEMERGENCY,ErrNULL,ADR(CmdExe),ADR(State),ADR(Error),ADR(ErrorLog));
					RegistroAlarma2205 := 32 ;
				END_IF	
				
				IF Ax^.Status.ErrorID <> ErrNULL THEN
					TFError(ErrAXIS,Ax^.Status.ErrorID,ADR(CmdExe),ADR(State),ADR(Error),ADR(ErrorLog));
				END_IF
				
			(* Case 13 - Attesa completamento comando *)	
			13:
				TFTimerSet(ADR(TempoFiltroTastatoriOFF),10,Px_Touch);
				IF Ax^.Status.MoveAbsoluteDone THEN
					Ax^.Command.MoveAbsolute := FALSE;
					TFCommandCase(ADR(CmdExe),100,CommandCase_JMP);
				ELSIF  Ax^.Status.MoveAbsoluteDone OR (NOT Programma^.DisabilitaTasteggio AND (NOT Px_Touch) AND TFTimerDone(ADR(TempoFiltroTastatoriOFF))) THEN  
					Ax^.Command.MoveAbsolute := FALSE;
					TFCommandCase(ADR(CmdExe),1,CommandCase_INC);
				ELSIF IN.Enable_TouchEmergency^ AND (NOT Px_TouchEmergency) THEN  
					Ax^.Command.MoveAbsolute := FALSE;
					TFError(ErrTOUCHEMERGENCY,ErrNULL,ADR(CmdExe),ADR(State),ADR(Error),ADR(ErrorLog));
					RegistroAlarma2205 := 33 ;
				ELSIF Ax^.Status.ErrorID <> ErrNULL THEN
					Ax^.Command.MoveAbsolute := FALSE;
					TFError(ErrAXIS,Ax^.Status.ErrorID,ADR(CmdExe),ADR(State),ADR(Error),ADR(ErrorLog));
				ELSIF TFTimerDone(ADR(Timeout))THEN
					Ax^.Command.MoveAbsolute := FALSE;
					TFError(ErrTOMOVE,ErrNULL,ADR(CmdExe),ADR(State),ADR(Error),ADR(ErrorLog));
				END_IF
				
